KUKA KRL program: MyProgram_031().src

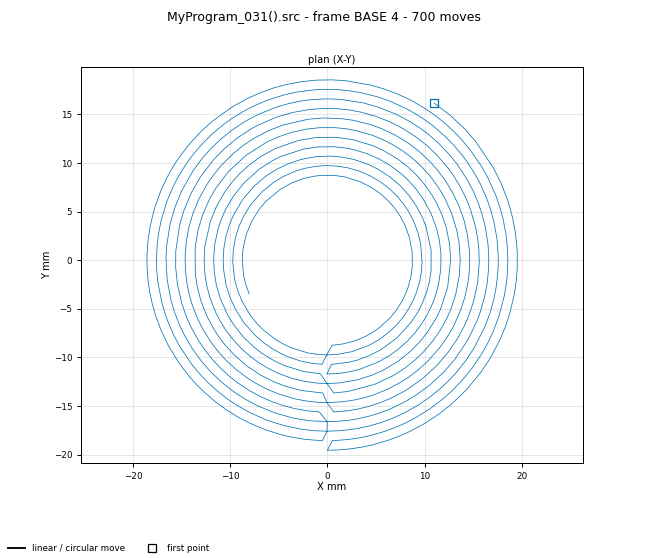
[picture p0: tool path of MyProgram_031().src in frame BASE 4, 700 of 700 moves have a stored position in this frame; points joined in program order, loops and branches not executed]
&ACCESS RVP
&REL 1
&PARAM TEMPLATE = C:\KRC\Roboter\Template\vorgabe
&PARAM EDITMASK = *
DEF MyProgram_031()
; ---- Setting reference (Base) ----
$BASE = BASE_DATA[4]

; --------------------------
; ---- Setting tool (TCP) ----
$TOOL = TOOL_DATA[3]
; --------------------------

$VEL.CP = VEL_APROX_PRINT
Startdeposition()
$VEL.CP = VEL_PRINT
LIN {X 10.9934,Y 16.1646,Z 59,A 46.5533,B 24.7923,C -3.3229,E1 25.0931,E2 -684.1777} C_DIS
LIN {X 12.5371,Y 14.9988,Z 59,A 41.0137,B 24.7934,C -3.3139,E1 25.1052,E2 -678.6373} C_DIS
LIN {X 14.028,Y 13.6149,Z 59,A 34.9278,B 24.795,C -3.3008,E1 25.1174,E2 -672.5458} C_DIS
LIN {X 15.29,Y 12.1806,Z 59,A 28.493,B 24.7975,C -3.281,E1 25.1289,E2 -666.0937} C_DIS
LIN {X 17.0834,Y 9.5029,Z 59,A 20.9449,B 24.7984,C -3.2739,E1 25.1402,E2 -658.5668} C_DIS
LIN {X 17.8595,Y 7.9485,Z 59,A 14.4237,B 24.8017,C -3.2472,E1 25.148,E2 -652.0173} C_DIS
LIN {X 18.5084,Y 6.2918,Z 59,A 10.2599,B 24.8023,C -3.2419,E1 25.152,E2 -647.8642} C_DIS
LIN {X 18.8302,Y 5.2505,Z 59,A 7.0393,B 24.8035,C -3.2323,E1 25.1545,E2 -644.6393} C_DIS
LIN {X 19.0668,Y 4.3128,Z 59,A 3.787,B 24.805,C -3.22,E1 25.1566,E2 -641.3766} C_DIS
LIN {X 19.331,Y 2.9059,Z 59,A 0.1157,B 24.806,C -3.2121,E1 25.1583,E2 -637.7083} C_DIS
LIN {X 19.4777,Y 1.6618,Z 59,A -3.1967,B 24.8069,C -3.2042,E1 25.1593,E2 -634.3968} C_DIS
LIN {X 19.5336,Y 0.7644,Z 59,A -6.4456,B 24.8086,C -3.1903,E1 25.1597,E2 -631.1341} C_DIS
LIN {X 19.5284,Y -0.889,Z 59,A -10.5652,B 24.8096,C -3.182,E1 25.1596,E2 -627.0194} C_DIS
LIN {X 19.4419,Y -2.0395,Z 59,A -14.3602,B 24.8113,C -3.1676,E1 25.1586,E2 -623.2127} C_DIS
LIN {X 19.2406,Y -3.4554,Z 59,A -19.2929,B 24.8137,C -3.1476,E1 25.1564,E2 -618.2616} C_DIS
LIN {X 18.7455,Y -5.5452,Z 59,A -24.8888,B 24.8152,C -3.1348,E1 25.1525,E2 -612.6677} C_DIS
LIN {X 18.3078,Y -6.8534,Z 59,A -28.9539,B 24.8167,C -3.1224,E1 25.1487,E2 -608.596} C_DIS
LIN {X 17.7883,Y -8.1069,Z 59,A -33.3998,B 24.8186,C -3.1064,E1 25.1437,E2 -604.1364} C_DIS
LIN {X 16.7634,Y -10.0571,Z 59,A -39.0828,B 24.8199,C -3.0952,E1 25.136,E2 -598.4565} C_DIS
LIN {X 15.7922,Y -11.5219,Z 59,A -45.0383,B 24.8223,C -3.0741,E1 25.1265,E2 -592.4803} C_DIS
LIN {X 14.2679,Y -13.3632,Z 59,A -52.0299,B 24.8243,C -3.0568,E1 25.1136,E2 -585.4791} C_DIS
LIN {X 12.7755,Y -14.7963,Z 59,A -57.4268,B 24.8253,C -3.0488,E1 25.1025,E2 -580.085} C_DIS
LIN {X 11.5072,Y -15.803,Z 59,A -62.4088,B 24.8266,C -3.037,E1 25.0914,E2 -575.0932} C_DIS
LIN {X 9.973,Y -16.8133,Z 59,A -67.5385,B 24.8275,C -3.0291,E1 25.0793,E2 -569.9612} C_DIS
LIN {X 8.5686,Y -17.5705,Z 59,A -72.3693,B 24.8285,C -3.0203,E1 25.0673,E2 -565.1228} C_DIS
LIN {X 7.4388,Y -18.0777,Z 59,A -75.5292,B 24.8287,C -3.0187,E1 25.0592,E2 -561.9667} C_DIS
LIN {X 6.3063,Y -18.5035,Z 59,A -79.4929,B 24.8296,C -3.0111,E1 25.0488,E2 -557.9929} C_DIS
LIN {X 4.7039,Y -18.9743,Z 59,A -83.9715,B 24.8298,C -3.009,E1 25.0367,E2 -553.5168} C_DIS
LIN {X 3.7008,Y -19.195,Z 59,A -86.9714,B 24.8301,C -3.0065,E1 25.0285,E2 -550.5147} C_DIS
LIN {X 2.5135,Y -19.3863,Z 59,A -90.6996,B 24.8305,C -3.0027,E1 25.0182,E2 -546.7808} C_DIS
LIN {X 1.1875,Y -19.5124,Z 59,A -94.7053,B 24.8308,C -3.0002,E1 25.007,E2 -542.7711} C_DIS
LIN {X -0.014,Y -19.5462,Z 59,A -96.7565,B 24.8298,C -3.0091,E1 25.0014,E2 -540.7413} C_DIS
Enddeposition()
LIN {X -0.014,Y -19.5462,Z 59,A -96.7565,B 24.8298,C -3.0091,E1 25.0014,E2 -540.7413} C_DIS
Startdeposition()
$VEL.CP = VEL_PRINT
LIN {X 0.5237,Y -18.5604,Z 59,A -93.787,B 24.8269,C -3.035,E1 25.0098,E2 -543.772} C_DIS
LIN {X 2.1884,Y -18.4383,Z 59,A -89.5474,B 24.8272,C -3.0316,E1 25.0216,E2 -548.0007} C_DIS
LIN {X 3.3621,Y -18.2608,Z 59,A -86.0615,B 24.8271,C -3.033,E1 25.0312,E2 -551.4866} C_DIS
LIN {X 4.4772,Y -18.0199,Z 59,A -81.9917,B 24.8263,C -3.0402,E1 25.0423,E2 -555.5678} C_DIS
LIN {X 5.9095,Y -17.6007,Z 59,A -77.975,B 24.8261,C -3.0412,E1 25.053,E2 -559.5795} C_DIS
LIN {X 7.3368,Y -17.0569,Z 59,A -73.4193,B 24.8256,C -3.0463,E1 25.0648,E2 -564.1373} C_DIS
LIN {X 8.1484,Y -16.6843,Z 59,A -70.3831,B 24.8248,C -3.0528,E1 25.0725,E2 -567.1809} C_DIS
LIN {X 9.0499,Y -16.213,Z 59,A -66.8043,B 24.8238,C -3.0616,E1 25.0813,E2 -570.7702} C_DIS
LIN {X 10.5141,Y -15.3044,Z 59,A -61.4455,B 24.8226,C -3.0719,E1 25.0938,E2 -576.1361} C_DIS
LIN {X 11.669,Y -14.4426,Z 59,A -57.2471,B 24.8218,C -3.0792,E1 25.1031,E2 -580.3362} C_DIS
LIN {X 12.719,Y -13.5275,Z 59,A -53.0786,B 24.8208,C -3.0878,E1 25.1117,E2 -584.5083} C_DIS
LIN {X 13.8411,Y -12.3769,Z 59,A -47.8137,B 24.819,C -3.1025,E1 25.1218,E2 -589.785} C_DIS
LIN {X 14.8798,Y -11.1066,Z 59,A -42.8261,B 24.8176,C -3.1149,E1 25.1303,E2 -594.7786} C_DIS
LIN {X 15.8537,Y -9.6656,Z 59,A -37.7384,B 24.8161,C -3.1271,E1 25.138,E2 -599.8697} C_DIS
LIN {X 16.5051,Y -8.5047,Z 59,A -33.7941,B 24.8149,C -3.1373,E1 25.1433,E2 -603.8175} C_DIS
LIN {X 17.0454,Y -7.3631,Z 59,A -29.7118,B 24.8134,C -3.1504,E1 25.148,E2 -607.9086} C_DIS
LIN {X 17.6434,Y -5.7852,Z 59,A -23.9683,B 24.8109,C -3.1711,E1 25.1533,E2 -613.6688} C_DIS
LIN {X 18.2032,Y -3.6604,Z 59,A -17.5312,B 24.8088,C -3.1887,E1 25.1574,E2 -620.1104} C_DIS
LIN {X 18.4301,Y -2.258,Z 59,A -13.7246,B 24.8078,C -3.197,E1 25.1589,E2 -623.9142} C_DIS
LIN {X 18.5284,Y -1.2107,Z 59,A -10.5836,B 24.8067,C -3.2061,E1 25.1596,E2 -627.0582} C_DIS
LIN {X 18.5698,Y -0.0273,Z 59,A -6.3825,B 24.8047,C -3.2226,E1 25.1597,E2 -631.2734} C_DIS
LIN {X 18.5205,Y 1.3276,Z 59,A -2.3554,B 24.8033,C -3.2341,E1 25.1591,E2 -635.3039} C_DIS
LIN {X 18.3716,Y 2.6925,Z 59,A 1.9622,B 24.8016,C -3.2478,E1 25.1575,E2 -639.6284} C_DIS
LIN {X 18.075,Y 4.2502,Z 59,A 6.671,B 24.8,C -3.2608,E1 25.1548,E2 -644.3406} C_DIS
LIN {X 17.7604,Y 5.4158,Z 59,A 10.2503,B 24.7988,C -3.2704,E1 25.152,E2 -647.9222} C_DIS
LIN {X 17.3583,Y 6.5919,Z 59,A 14.5526,B 24.7969,C -3.2855,E1 25.1478,E2 -652.2364} C_DIS
LIN {X 16.5083,Y 8.4991,Z 59,A 20.2918,B 24.7955,C -3.2968,E1 25.141,E2 -657.9714} C_DIS
LIN {X 15.8062,Y 9.7434,Z 59,A 25.4816,B 24.7933,C -3.315,E1 25.1335,E2 -663.1777} C_DIS
LIN {X 14.5876,Y 11.4876,Z 59,A 31.3946,B 24.792,C -3.325,E1 25.1238,E2 -669.0861} C_DIS
LIN {X 13.6613,Y 12.575,Z 59,A 35.618,B 24.791,C -3.3332,E1 25.116,E2 -673.3099} C_DIS
LIN {X 12.7974,Y 13.4532,Z 59,A 39.7636,B 24.7896,C -3.3437,E1 25.1077,E2 -677.4632} C_DIS
LIN {X 11.9589,Y 14.2042,Z 59,A 43.058,B 24.789,C -3.3488,E1 25.1007,E2 -680.7568} C_DIS
LIN {X 11.0207,Y 14.9437,Z 59,A 46.3495,B 24.7886,C -3.3521,E1 25.0934,E2 -684.0441} C_DIS
LIN {X 9.9784,Y 15.6588,Z 59,A 50.7011,B 24.7874,C -3.3616,E1 25.0833,E2 -688.4039} C_DIS
LIN {X 8.6913,Y 16.4082,Z 59,A 55.2475,B 24.7866,C -3.3674,E1 25.0722,E2 -692.9507} C_DIS
LIN {X 7.4621,Y 17.0024,Z 59,A 59.3101,B 24.7862,C -3.371,E1 25.0619,E2 -697.0117} C_DIS
LIN {X 5.9289,Y 17.5955,Z 59,A 64.5931,B 24.7854,C -3.377,E1 25.048,E2 -702.2978} C_DIS
LIN {X 4.4746,Y 18.0207,Z 59,A 69.9369,B 24.7845,C -3.3843,E1 25.0335,E2 -707.6509} C_DIS
LIN {X 1.7966,Y 18.4808,Z 59,A 77.036,B 24.7852,C -3.3783,E1 25.014,E2 -714.7291} C_DIS
LIN {X 0.4664,Y 18.562,Z 59,A 81.8933,B 24.7847,C -3.3825,E1 25.0004,E2 -719.5951} C_DIS
LIN {X -1.1715,Y 18.5307,Z 59,A 86.5563,B 24.7852,C -3.3787,E1 24.9874,E2 -724.2497} C_DIS
LIN {X -2.6397,Y 18.3778,Z 59,A 90.8462,B 24.7857,C -3.3747,E1 24.9756,E2 -728.533} C_DIS
LIN {X -4.1478,Y 18.0986,Z 59,A 96.1737,B 24.7857,C -3.374,E1 24.961,E2 -733.865} C_DIS
LIN {X -5.4949,Y 17.7361,Z 59,A 100.4335,B 24.7864,C -3.3692,E1 24.9496,E2 -738.1204} C_DIS
LIN {X -7.0138,Y 17.1921,Z 59,A 105.1464,B 24.7874,C -3.3615,E1 24.9373,E2 -742.8249} C_DIS
LIN {X -8.3436,Y 16.5877,Z 59,A 110.1725,B 24.7879,C -3.3571,E1 24.9246,E2 -747.8532} C_DIS
LIN {X -9.8622,Y 15.7322,Z 59,A 115.7778,B 24.789,C -3.3486,E1 24.9112,E2 -753.4554} C_DIS
LIN {X -11.794,Y 14.3412,Z 59,A 122.0514,B 24.7915,C -3.3294,E1 24.8973,E2 -759.7053} C_DIS
LIN {X -12.9768,Y 13.2796,Z 59,A 128.0289,B 24.7923,C -3.3224,E1 24.885,E2 -765.6906} C_DIS
LIN {X -14.3419,Y 11.7922,Z 59,A 134.5147,B 24.7941,C -3.3079,E1 24.8732,E2 -772.1711} C_DIS
LIN {X -15.524,Y 10.1868,Z 59,A 139.7208,B 24.7966,C -3.2883,E1 24.8649,E2 -777.3557} C_DIS
LIN {X -16.0114,Y 9.4022,Z 59,A 142.6599,B 24.7975,C -3.2807,E1 24.8607,E2 -780.2918} C_DIS
LIN {X -16.5699,Y 8.3788,Z 59,A 146.5868,B 24.7987,C -3.2715,E1 24.8556,E2 -784.2176} C_DIS
LIN {X -17.1414,Y 7.1369,Z 59,A 150.9696,B 24.8001,C -3.2597,E1 24.8507,E2 -788.5962} C_DIS
LIN {X -17.7821,Y 5.3442,Z 59,A 157.1224,B 24.8022,C -3.2429,E1 24.8454,E2 -794.7439} C_DIS
LIN {X -18.2292,Y 3.5294,Z 59,A 162.1023,B 24.8047,C -3.2227,E1 24.8423,E2 -799.7047} C_DIS
LIN {X -18.4463,Y 2.1199,Z 59,A 167.1635,B 24.8061,C -3.211,E1 24.8404,E2 -804.7681} C_DIS
LIN {X -18.5634,Y 0.4029,Z 59,A 172.0002,B 24.8083,C -3.1931,E1 24.8398,E2 -809.5908} C_DIS
LIN {X -18.5529,Y -0.7461,Z 59,A 175.4062,B 24.8096,C -3.1816,E1 24.84,E2 -812.99} C_DIS
LIN {X -18.4568,Y -2.027,Z 59,A 179.3572,B 24.8111,C -3.1694,E1 24.8409,E2 -816.9354} C_DIS
LIN {X -18.3051,Y -3.1127,Z 59,A -176.6587,B 24.8121,C -3.161,E1 24.8427,E2 -820.923} C_DIS
LIN {X -18.0102,Y -4.5166,Z 59,A -172.3898,B 24.8137,C -3.1473,E1 24.8453,E2 -825.1841} C_DIS
LIN {X -17.6745,Y -5.69,Z 59,A -168.215,B 24.8149,C -3.1377,E1 24.8488,E2 -829.3599} C_DIS
LIN {X -17.09,Y -7.2591,Z 59,A -163.1852,B 24.8167,C -3.1227,E1 24.854,E2 -834.3819} C_DIS
LIN {X -16.3676,Y -8.7671,Z 59,A -158.089,B 24.8183,C -3.1086,E1 24.8604,E2 -839.4719} C_DIS
LIN {X -15.3002,Y -10.52,Z 59,A -150.8716,B 24.8198,C -3.0961,E1 24.8713,E2 -846.6957} C_DIS
LIN {X -14.1699,Y -11.9992,Z 59,A -146.4366,B 24.8219,C -3.0779,E1 24.879,E2 -851.1077} C_DIS
LIN {X -13.5514,Y -12.6934,Z 59,A -142.9303,B 24.8223,C -3.0743,E1 24.8857,E2 -854.6209} C_DIS
LIN {X -12.6198,Y -13.6202,Z 59,A -138.756,B 24.8232,C -3.0667,E1 24.8941,E2 -858.7944} C_DIS
LIN {X -11.4375,Y -14.6271,Z 59,A -134.7068,B 24.8246,C -3.0549,E1 24.9028,E2 -862.8306} C_DIS
LIN {X -10.4429,Y -15.3528,Z 59,A -130.1092,B 24.8249,C -3.0524,E1 24.9133,E2 -867.438} C_DIS
LIN {X -9.2262,Y -16.1134,Z 59,A -126.1346,B 24.8258,C -3.044,E1 24.9228,E2 -871.4047} C_DIS
LIN {X -8.0735,Y -16.7207,Z 59,A -121.9508,B 24.8263,C -3.04,E1 24.9333,E2 -875.5902} C_DIS
LIN {X -6.4151,Y -17.4242,Z 59,A -115.4888,B 24.8263,C -3.0396,E1 24.9501,E2 -882.0652} C_DIS
LIN {X -4.7827,Y -17.9413,Z 59,A -111.2767,B 24.8274,C -3.0302,E1 24.9613,E2 -886.2617} C_DIS
LIN {X -3.7911,Y -18.1762,Z 59,A -108.016,B 24.8274,C -3.0294,E1 24.9702,E2 -889.5247} C_DIS
LIN {X -2.2382,Y -18.4325,Z 59,A -102.9506,B 24.8274,C -3.0296,E1 24.9842,E2 -894.5947} C_DIS
LIN {X -0.5182,Y -18.5594,Z 59,A -97.8029,B 24.8276,C -3.0288,E1 24.9986,E2 -899.742} C_DIS
LIN {X -0.5182,Y -18.5594,Z 59,A -97.8029,B 24.8276,C -3.0288,E1 24.9986,E2 -899.742} C_DIS
Enddeposition()
LIN {X -0.0341,Y -17.5871,Z 59,A -98.1601,B 24.8269,C -3.0347,E1 24.9976,E2 -899.3987} C_DIS
Startdeposition()
$VEL.CP = VEL_PRINT
LIN {X -1.202,Y -17.546,Z 59,A -102.1315,B 24.827,C -3.0335,E1 24.9865,E2 -895.4234} C_DIS
LIN {X -2.6082,Y -17.3925,Z 59,A -107.1397,B 24.8272,C -3.0321,E1 24.9726,E2 -890.4083} C_DIS
LIN {X -4.5044,Y -17.0004,Z 59,A -113.0275,B 24.8266,C -3.0373,E1 24.9566,E2 -884.5252} C_DIS
LIN {X -6.2144,Y -16.4525,Z 59,A -119.7875,B 24.8266,C -3.0376,E1 24.9388,E2 -877.753} C_DIS
LIN {X -7.9886,Y -15.6679,Z 59,A -125.5503,B 24.8254,C -3.0473,E1 24.9243,E2 -871.9985} C_DIS
LIN {X -9.3669,Y -14.8852,Z 59,A -130.316,B 24.8244,C -3.0562,E1 24.9129,E2 -867.2397} C_DIS
LIN {X -10.2976,Y -14.2571,Z 59,A -133.7611,B 24.8236,C -3.0629,E1 24.905,E2 -863.7988} C_DIS
LIN {X -11.2418,Y -13.5251,Z 59,A -138.3974,B 24.8232,C -3.0669,E1 24.8949,E2 -859.1548} C_DIS
LIN {X -12.4133,Y -12.4588,Z 59,A -143.1705,B 24.8218,C -3.0785,E1 24.8852,E2 -854.3898} C_DIS
LIN {X -13.276,Y -11.5347,Z 59,A -147.4681,B 24.8209,C -3.0868,E1 24.8772,E2 -850.093} C_DIS
LIN {X -14.0207,Y -10.6174,Z 59,A -152.0625,B 24.8201,C -3.0934,E1 24.8693,E2 -845.4924} C_DIS
LIN {X -15.21,Y -8.8298,Z 59,A -158.0938,B 24.8177,C -3.1139,E1 24.8604,E2 -839.4797} C_DIS
LIN {X -15.8554,Y -7.6095,Z 59,A -162.9618,B 24.8164,C -3.1249,E1 24.8542,E2 -834.6118} C_DIS
LIN {X -16.5043,Y -6.0742,Z 59,A -169.1979,B 24.8149,C -3.1379,E1 24.8479,E2 -828.3721} C_DIS
LIN {X -16.9974,Y -4.5159,Z 59,A -174.5907,B 24.813,C -3.1534,E1 24.8438,E2 -822.985} C_DIS
LIN {X -17.4451,Y -2.2294,Z 59,A 179.1035,B 24.8099,C -3.1797,E1 24.8409,E2 -816.7048} C_DIS
LIN {X -17.5572,Y -1.0226,Z 59,A 175.2609,B 24.8084,C -3.1921,E1 24.84,E2 -812.8688} C_DIS
LIN {X -17.5889,Y -0.0438,Z 59,A 170.9905,B 24.8075,C -3.1993,E1 24.8398,E2 -808.59} C_DIS
LIN {X -17.5028,Y 1.7202,Z 59,A 165.8261,B 24.8052,C -3.2187,E1 24.8408,E2 -803.441} C_DIS
LIN {X -17.3482,Y 2.8889,Z 59,A 161.8878,B 24.8037,C -3.2303,E1 24.8424,E2 -799.5072} C_DIS
LIN {X -17.1003,Y 4.1084,Z 59,A 157.2587,B 24.8024,C -3.2414,E1 24.8453,E2 -794.8774} C_DIS
LIN {X -16.5111,Y 6.057,Z 59,A 150.2732,B 24.8,C -3.2604,E1 24.8515,E2 -787.8977} C_DIS
LIN {X -15.838,Y 7.646,Z 59,A 145.3885,B 24.7978,C -3.2787,E1 24.8571,E2 -783.0302} C_DIS
LIN {X -15.2784,Y 8.7108,Z 59,A 141.3244,B 24.7965,C -3.2894,E1 24.8625,E2 -778.9702} C_DIS
LIN {X -14.5545,Y 9.8727,Z 59,A 137.2092,B 24.7948,C -3.3025,E1 24.8688,E2 -774.8656} C_DIS
LIN {X -13.9706,Y 10.683,Z 59,A 133.478,B 24.7939,C -3.3095,E1 24.875,E2 -771.1334} C_DIS
LIN {X -13,Y 11.8452,Z 59,A 128.5098,B 24.7924,C -3.3216,E1 24.8841,E2 -766.1716} C_DIS
LIN {X -11.8535,Y 12.9918,Z 59,A 123.7688,B 24.7907,C -3.3355,E1 24.8936,E2 -761.4442} C_DIS
LIN {X -10.7852,Y 13.892,Z 59,A 119.0842,B 24.7895,C -3.3447,E1 24.9037,E2 -756.7638} C_DIS
LIN {X -9.7714,Y 14.623,Z 59,A 114.5567,B 24.7887,C -3.3509,E1 24.9141,E2 -752.2359} C_DIS
LIN {X -8.6558,Y 15.3098,Z 59,A 110.5552,B 24.7877,C -3.3594,E1 24.9237,E2 -748.2425} C_DIS
LIN {X -7.5105,Y 15.9027,Z 59,A 106.0225,B 24.787,C -3.3646,E1 24.935,E2 -743.7103} C_DIS
LIN {X -6.2319,Y 16.4459,Z 59,A 101.4023,B 24.7863,C -3.3702,E1 24.947,E2 -739.0934} C_DIS
LIN {X -4.4803,Y 17.0067,Z 59,A 96.1433,B 24.785,C -3.3799,E1 24.961,E2 -733.8488} C_DIS
LIN {X -3.1544,Y 17.3018,Z 59,A 90.8771,B 24.785,C -3.3795,E1 24.9754,E2 -728.5754} C_DIS
LIN {X -1.3631,Y 17.534,Z 59,A 85.5279,B 24.7843,C -3.3853,E1 24.9903,E2 -723.2369} C_DIS
LIN {X -0.2748,Y 17.585,Z 59,A 81.8951,B 24.7843,C -3.3859,E1 25.0004,E2 -719.605} C_DIS
LIN {X 0.9445,Y 17.5616,Z 59,A 77.9768,B 24.7842,C -3.3865,E1 25.0113,E2 -715.6891} C_DIS
LIN {X 2.0251,Y 17.4701,Z 59,A 74.5767,B 24.7842,C -3.3869,E1 25.0208,E2 -712.292} C_DIS
LIN {X 3.3851,Y 17.2583,Z 59,A 69.3654,B 24.7849,C -3.381,E1 25.0351,E2 -707.0723} C_DIS
LIN {X 5.1414,Y 16.8186,Z 59,A 63.7363,B 24.7852,C -3.3789,E1 25.0503,E2 -701.4474} C_DIS
LIN {X 6.5268,Y 16.3312,Z 59,A 58.7341,B 24.7859,C -3.3731,E1 25.0633,E2 -696.4421} C_DIS
LIN {X 8.2661,Y 15.5236,Z 59,A 52.7014,B 24.7867,C -3.3671,E1 25.0784,E2 -690.4112} C_DIS
LIN {X 9.239,Y 14.9649,Z 59,A 49.4605,B 24.787,C -3.3648,E1 25.0862,E2 -687.1748} C_DIS
LIN {X 10.1074,Y 14.3927,Z 59,A 46.1864,B 24.7875,C -3.3602,E1 25.0937,E2 -683.901} C_DIS
LIN {X 10.8842,Y 13.8142,Z 59,A 42.5638,B 24.7887,C -3.3513,E1 25.1018,E2 -680.2704} C_DIS
LIN {X 12.1818,Y 12.685,Z 59,A 36.9397,B 24.7901,C -3.3402,E1 25.1134,E2 -674.6427} C_DIS
LIN {X 13.0558,Y 11.7832,Z 59,A 33.0738,B 24.791,C -3.3332,E1 25.1207,E2 -670.7771} C_DIS
LIN {X 13.8849,Y 10.7944,Z 59,A 29.1416,B 24.7919,C -3.3258,E1 25.1276,E2 -666.8454} C_DIS
LIN {X 14.4707,Y 9.9948,Z 59,A 25.5134,B 24.7933,C -3.3147,E1 25.1335,E2 -663.2087} C_DIS
LIN {X 15.296,Y 8.6798,Z 59,A 20.8881,B 24.7945,C -3.3053,E1 25.1402,E2 -658.5848} C_DIS
LIN {X 15.7748,Y 7.7754,Z 59,A 17.229,B 24.7959,C -3.2937,E1 25.1448,E2 -654.9175} C_DIS
LIN {X 16.3754,Y 6.4149,Z 59,A 12.8077,B 24.7972,C -3.2837,E1 25.1496,E2 -650.4969} C_DIS
LIN {X 16.7585,Y 5.3277,Z 59,A 9.1385,B 24.7984,C -3.2737,E1 25.1529,E2 -646.8246} C_DIS
LIN {X 17.1612,Y 3.847,Z 59,A 3.5488,B 24.8009,C -3.2537,E1 25.1567,E2 -641.2198} C_DIS
LIN {X 17.4561,Y 2.1435,Z 59,A -2.1885,B 24.8031,C -3.2357,E1 25.159,E2 -635.4734} C_DIS
LIN {X 17.5829,Y 0.389,Z 59,A -7.321,B 24.8046,C -3.2232,E1 25.1598,E2 -630.3418} C_DIS
LIN {X 17.5693,Y -0.791,Z 59,A -11.7704,B 24.8067,C -3.2059,E1 25.1594,E2 -625.8779} C_DIS
LIN {X 17.3971,Y -2.5796,Z 59,A -17.0839,B 24.8083,C -3.1924,E1 25.1576,E2 -620.5638} C_DIS
LIN {X 17.1448,Y -3.9184,Z 59,A -21.4856,B 24.81,C -3.179,E1 25.1551,E2 -616.156} C_DIS
LIN {X 16.7502,Y -5.3608,Z 59,A -26.9183,B 24.8123,C -3.1593,E1 25.1507,E2 -610.7076} C_DIS
LIN {X 16.2207,Y -6.7963,Z 59,A -32.3118,B 24.8145,C -3.141,E1 25.1451,E2 -605.3005} C_DIS
LIN {X 15.1393,Y -8.9502,Z 59,A -39.1864,B 24.8162,C -3.127,E1 25.136,E2 -598.4287} C_DIS
LIN {X 14.2994,Y -10.2387,Z 59,A -43.7759,B 24.8173,C -3.1169,E1 25.1288,E2 -593.8382} C_DIS
LIN {X 13.3413,Y -11.4595,Z 59,A -48.9758,B 24.819,C -3.1028,E1 25.1196,E2 -588.6289} C_DIS
LIN {X 12.4978,Y -12.3738,Z 59,A -53.1294,B 24.8202,C -3.0922,E1 25.1116,E2 -584.4683} C_DIS
LIN {X 11.523,Y -13.2864,Z 59,A -57.5824,B 24.8215,C -3.0816,E1 25.1024,E2 -580.0079} C_DIS
LIN {X 10.5304,Y -14.0857,Z 59,A -61.3966,B 24.8222,C -3.0756,E1 25.0939,E2 -576.1935} C_DIS
LIN {X 9.3514,Y -14.8949,Z 59,A -66.5114,B 24.8236,C -3.0633,E1 25.082,E2 -571.0663} C_DIS
LIN {X 7.881,Y -15.7225,Z 59,A -71.8747,B 24.8245,C -3.0551,E1 25.0688,E2 -565.6989} C_DIS
LIN {X 6.6785,Y -16.2696,Z 59,A -75.7384,B 24.8249,C -3.052,E1 25.0589,E2 -561.8372} C_DIS
LIN {X 5.5387,Y -16.6921,Z 59,A -79.5762,B 24.8254,C -3.0479,E1 25.0488,E2 -557.9973} C_DIS
LIN {X 4.3173,Y -17.049,Z 59,A -84.2933,B 24.8263,C -3.0397,E1 25.036,E2 -553.2684} C_DIS
LIN {X 3.067,Y -17.3175,Z 59,A -88.4641,B 24.8267,C -3.0363,E1 25.0246,E2 -549.0944} C_DIS
LIN {X 1.512,Y -17.5221,Z 59,A -93.4732,B 24.827,C -3.0341,E1 25.0107,E2 -544.0834} C_DIS
LIN {X -0.0341,Y -17.5871,Z 59,A -95.9822,B 24.8254,C -3.0478,E1 25.0038,E2 -541.6078} C_DIS
Enddeposition()
LIN {X -0.0167,Y -16.6038,Z 59,A -2.603,B -0.0001,C -0.0021,E1 0.1598,E2 -630.6872} C_DIS
Startdeposition()
$VEL.CP = VEL_PRINT
LIN {X 0.9904,Y -16.5764,Z 59,A -2.567,B -0.0002,C -0.0021,E1 0.1597,E2 -630.6857} C_DIS
LIN {X 2.1202,Y -16.4703,Z 59,A -2.5264,B -0.0004,C -0.0021,E1 0.1595,E2 -630.681} C_DIS
LIN {X 3.0555,Y -16.3228,Z 59,A -2.4952,B -0.0005,C -0.0021,E1 0.1594,E2 -630.6719} C_DIS
LIN {X 4.3685,Y -16.0213,Z 59,A -2.4467,B -0.0007,C -0.0021,E1 0.1592,E2 -630.6599} C_DIS
LIN {X 5.3661,Y -15.7154,Z 59,A -2.4124,B -0.0007,C -0.002,E1 0.1591,E2 -630.6448} C_DIS
LIN {X 6.4776,Y -15.2909,Z 59,A -2.3767,B -0.001,C -0.0019,E1 0.1589,E2 -630.6217} C_DIS
LIN {X 7.9833,Y -14.5611,Z 59,A -2.3219,B -0.0011,C -0.0018,E1 0.1587,E2 -630.59} C_DIS
LIN {X 9.1663,Y -13.8473,Z 59,A -2.2799,B -0.0013,C -0.0017,E1 0.1587,E2 -630.5578} C_DIS
LIN {X 10.5664,Y -12.8103,Z 59,A -2.2377,B -0.0015,C -0.0015,E1 0.1584,E2 -630.5035} C_DIS
LIN {X 12.0029,Y -11.4754,Z 59,A -2.1921,B -0.0016,C -0.0013,E1 0.1582,E2 -630.438} C_DIS
LIN {X 13.1246,Y -10.1742,Z 59,A -2.1569,B -0.0018,C -0.0012,E1 0.1581,E2 -630.375} C_DIS
LIN {X 14.4222,Y -8.2322,Z 59,A -2.1137,B -0.0019,C -0.0009,E1 0.1579,E2 -630.2853} C_DIS
LIN {X 15.3466,Y -6.3442,Z 59,A -2.0661,B -0.0019,C -0.0007,E1 0.1579,E2 -630.2164} C_DIS
LIN {X 15.729,Y -5.3263,Z 59,A -2.0674,B -0.002,C -0.0006,E1 0.1578,E2 -630.1562} C_DIS
LIN {X 16.1828,Y -3.7261,Z 59,A -2.0525,B -0.002,C -0.0004,E1 0.1578,E2 -630.0842} C_DIS
LIN {X 16.4301,Y -2.4133,Z 59,A -2.0455,B -0.0021,C -0.0002,E1 0.1577,E2 -630.0246} C_DIS
LIN {X 16.5743,Y -1.0125,Z 59,A -2.0396,B -0.0021,C 0,E1 0.1577,E2 -629.964} C_DIS
LIN {X 16.6055,Y 0.1927,Z 59,A -2.046,B -0.0021,C 0.0001,E1 0.1577,E2 -629.9038} C_DIS
LIN {X 16.5283,Y 1.6086,Z 59,A -2.0584,B -0.0021,C 0.0003,E1 0.1577,E2 -629.8325} C_DIS
LIN {X 16.2604,Y 3.3713,Z 59,A -2.0679,B -0.0021,C 0.0005,E1 0.1577,E2 -629.7563} C_DIS
LIN {X 15.9251,Y 4.7056,Z 59,A -2.0806,B -0.002,C 0.0007,E1 0.1577,E2 -629.6984} C_DIS
LIN {X 15.4863,Y 5.9956,Z 59,A -2.106,B -0.002,C 0.0009,E1 0.1578,E2 -629.6335} C_DIS
LIN {X 15.0367,Y 7.0473,Z 59,A -2.1262,B -0.0019,C 0.001,E1 0.1579,E2 -629.5847} C_DIS
LIN {X 14.3539,Y 8.3512,Z 59,A -2.1566,B -0.0018,C 0.0012,E1 0.1579,E2 -629.5237} C_DIS
LIN {X 13.351,Y 9.8748,Z 59,A -2.1863,B -0.0016,C 0.0013,E1 0.1581,E2 -629.4663} C_DIS
LIN {X 12.5968,Y 10.821,Z 59,A -2.227,B -0.0016,C 0.0015,E1 0.1582,E2 -629.4133} C_DIS
LIN {X 11.4808,Y 11.9985,Z 59,A -2.2698,B -0.0014,C 0.0016,E1 0.1584,E2 -629.3622} C_DIS
LIN {X 10.3808,Y 12.962,Z 59,A -2.3081,B -0.0012,C 0.0017,E1 0.1584,E2 -629.3243} C_DIS
LIN {X 9.587,Y 13.5597,Z 59,A -2.3443,B -0.0012,C 0.0018,E1 0.1586,E2 -629.2926} C_DIS
LIN {X 8.5013,Y 14.2653,Z 59,A -2.3855,B -0.001,C 0.0018,E1 0.1588,E2 -629.2625} C_DIS
LIN {X 7.0867,Y 15.0181,Z 59,A -2.4413,B -0.0008,C 0.002,E1 0.159,E2 -629.2281} C_DIS
LIN {X 5.2232,Y 15.7634,Z 59,A -2.5104,B -0.0005,C 0.002,E1 0.1592,E2 -629.198} C_DIS
LIN {X 3.6139,Y 16.2079,Z 59,A -2.5708,B -0.0003,C 0.002,E1 0.1594,E2 -629.1796} C_DIS
LIN {X 1.3286,Y 16.5531,Z 59,A -2.6524,B 0,C 0.0021,E1 0.1597,E2 -629.1697} C_DIS
LIN {X -0.0236,Y 16.6065,Z 59,A -2.7012,B 0.0002,C 0.0021,E1 0.1599,E2 -629.1697} C_DIS
LIN {X -1.5553,Y 16.5333,Z 59,A -2.7565,B 0.0003,C 0.0021,E1 0.16,E2 -629.1751} C_DIS
LIN {X -2.7667,Y 16.3742,Z 59,A -2.7997,B 0.0005,C 0.0021,E1 0.1602,E2 -629.1841} C_DIS
LIN {X -3.9498,Y 16.1297,Z 59,A -2.8411,B 0.0006,C 0.0021,E1 0.1603,E2 -629.1973} C_DIS
LIN {X -5.2286,Y 15.7615,Z 59,A -2.8832,B 0.0008,C 0.002,E1 0.1605,E2 -629.2184} C_DIS
LIN {X -7.1262,Y 14.9994,Z 59,A -2.9471,B 0.0011,C 0.0018,E1 0.1608,E2 -629.2574} C_DIS
LIN {X -8.4091,Y 14.3198,Z 59,A -2.993,B 0.0012,C 0.0018,E1 0.1609,E2 -629.2876} C_DIS
LIN {X -9.7953,Y 13.4097,Z 59,A -3.0364,B 0.0014,C 0.0016,E1 0.1611,E2 -629.3336} C_DIS
LIN {X -11.0607,Y 12.3867,Z 59,A -3.0781,B 0.0015,C 0.0015,E1 0.1613,E2 -629.3814} C_DIS
LIN {X -12.126,Y 11.3435,Z 59,A -3.1185,B 0.0016,C 0.0013,E1 0.1613,E2 -629.424} C_DIS
LIN {X -12.8622,Y 10.5035,Z 59,A -3.1341,B 0.0017,C 0.0013,E1 0.1615,E2 -629.4704} C_DIS
LIN {X -13.8438,Y 9.1716,Z 59,A -3.1593,B 0.0019,C 0.001,E1 0.1616,E2 -629.5367} C_DIS
LIN {X -15.0107,Y 7.1025,Z 59,A -3.1988,B 0.0019,C 0.0008,E1 0.1617,E2 -629.6261} C_DIS
LIN {X -15.7152,Y 5.3667,Z 59,A -3.2115,B 0.0021,C 0.0005,E1 0.1618,E2 -629.7112} C_DIS
LIN {X -16.1915,Y 3.6878,Z 59,A -3.2212,B 0.0021,C 0.0003,E1 0.1618,E2 -629.7887} C_DIS
LIN {X -16.5438,Y 1.437,Z 59,A -3.2403,B 0.0021,C 0,E1 0.1619,E2 -629.8763} C_DIS
LIN {X -16.6045,Y 0.2489,Z 59,A -3.2246,B 0.0021,C -0.0002,E1 0.1619,E2 -629.9436} C_DIS
LIN {X -16.4836,Y -2.0164,Z 59,A -3.2086,B 0.0021,C -0.0005,E1 0.1619,E2 -630.0497} C_DIS
LIN {X -16.0863,Y -4.1232,Z 59,A -3.2036,B 0.0021,C -0.0007,E1 0.1619,E2 -630.1286} C_DIS
LIN {X -15.7744,Y -5.1895,Z 59,A -3.1849,B 0.002,C -0.0008,E1 0.1618,E2 -630.1807} C_DIS
LIN {X -15.2365,Y -6.6046,Z 59,A -3.1653,B 0.0019,C -0.001,E1 0.1618,E2 -630.2404} C_DIS
LIN {X -14.7296,Y -7.6681,Z 59,A -3.1461,B 0.0019,C -0.0011,E1 0.1617,E2 -630.2861} C_DIS
LIN {X -13.908,Y -9.074,Z 59,A -3.1038,B 0.0017,C -0.0013,E1 0.1615,E2 -630.3581} C_DIS
LIN {X -12.9961,Y -10.3379,Z 59,A -3.0716,B 0.0016,C -0.0014,E1 0.1615,E2 -630.4109} C_DIS
LIN {X -12.0357,Y -11.4418,Z 59,A -3.0367,B 0.0014,C -0.0016,E1 0.1613,E2 -630.458} C_DIS
LIN {X -10.8435,Y -12.5767,Z 59,A -2.9901,B 0.0013,C -0.0017,E1 0.1611,E2 -630.5101} C_DIS
LIN {X -9.6701,Y -13.5004,Z 59,A -2.9454,B 0.0011,C -0.0018,E1 0.161,E2 -630.5519} C_DIS
LIN {X -8.4838,Y -14.2755,Z 59,A -2.9022,B 0.0009,C -0.0018,E1 0.1608,E2 -630.5856} C_DIS
LIN {X -7.2507,Y -14.9399,Z 59,A -2.8567,B 0.0008,C -0.002,E1 0.1607,E2 -630.6153} C_DIS
LIN {X -5.4913,Y -15.6721,Z 59,A -2.7899,B 0.0005,C -0.002,E1 0.1604,E2 -630.6503} C_DIS
LIN {X -3.7975,Y -16.1648,Z 59,A -2.7331,B 0.0004,C -0.002,E1 0.1603,E2 -630.6674} C_DIS
LIN {X -2.7555,Y -16.3761,Z 59,A -2.6949,B 0.0002,C -0.0021,E1 0.1601,E2 -630.6774} C_DIS
LIN {X -1.6353,Y -16.5256,Z 59,A -2.6548,B 0.0001,C -0.0021,E1 0.16,E2 -630.6836} C_DIS
LIN {X -0.0167,Y -16.6038,Z 59,A -2.5969,B -0.0001,C -0.0021,E1 0.1598,E2 -630.6867} C_DIS
Enddeposition()
LIN {X -0.0167,Y -16.6038,Z 59,A -2.5969,B -0.0001,C -0.0021,E1 0.1598,E2 -630.6867} C_DIS
Startdeposition()
$VEL.CP = VEL_PRINT
LIN {X -0.8365,Y -15.6031,Z 59,A -2.5752,B 0.0001,C -0.0021,E1 0.16,E2 -630.6942} C_DIS
LIN {X -2.0793,Y -15.4866,Z 59,A -2.6239,B 0.0002,C -0.0021,E1 0.1601,E2 -630.6852} C_DIS
LIN {X -3.4213,Y -15.2464,Z 59,A -2.673,B 0.0004,C -0.0021,E1 0.1603,E2 -630.6739} C_DIS
LIN {X -4.4197,Y -14.9875,Z 59,A -2.7127,B 0.0005,C -0.0021,E1 0.1604,E2 -630.659} C_DIS
LIN {X -5.5531,Y -14.6054,Z 59,A -2.758,B 0.0007,C -0.0021,E1 0.1606,E2 -630.638} C_DIS
LIN {X -6.8076,Y -14.0647,Z 59,A -2.8065,B 0.0009,C -0.002,E1 0.1608,E2 -630.6113} C_DIS
LIN {X -7.9948,Y -13.4253,Z 59,A -2.8587,B 0.0011,C -0.0019,E1 0.1609,E2 -630.5743} C_DIS
LIN {X -9.1231,Y -12.6858,Z 59,A -2.902,B 0.0011,C -0.0018,E1 0.1611,E2 -630.5401} C_DIS
LIN {X -10.0197,Y -11.9902,Z 59,A -2.9405,B 0.0013,C -0.0017,E1 0.1612,E2 -630.5041} C_DIS
LIN {X -10.8903,Y -11.2055,Z 59,A -2.98,B 0.0015,C -0.0016,E1 0.1613,E2 -630.4625} C_DIS
LIN {X -11.8306,Y -10.2076,Z 59,A -3.0202,B 0.0015,C -0.0014,E1 0.1614,E2 -630.4138} C_DIS
LIN {X -12.707,Y -9.0935,Z 59,A -3.0619,B 0.0017,C -0.0013,E1 0.1616,E2 -630.3565} C_DIS
LIN {X -13.3249,Y -8.1614,Z 59,A -3.0891,B 0.0017,C -0.0012,E1 0.1616,E2 -630.3122} C_DIS
LIN {X -13.997,Y -6.9453,Z 59,A -3.1227,B 0.0019,C -0.001,E1 0.1617,E2 -630.2515} C_DIS
LIN {X -14.5067,Y -5.8063,Z 59,A -3.1431,B 0.0019,C -0.0009,E1 0.1617,E2 -630.2017} C_DIS
LIN {X -14.9859,Y -4.4244,Z 59,A -3.1875,B 0.002,C -0.0006,E1 0.1619,E2 -630.1167} C_DIS
LIN {X -15.4335,Y -2.4391,Z 59,A -3.2009,B 0.0021,C -0.0004,E1 0.1619,E2 -630.0361} C_DIS
LIN {X -15.6083,Y -0.7284,Z 59,A -3.2373,B 0.0021,C -0.0001,E1 0.1619,E2 -629.9348} C_DIS
LIN {X -15.5966,Y 0.9527,Z 59,A -3.2485,B 0.0021,C 0.0001,E1 0.1619,E2 -629.853} C_DIS
LIN {X -15.208,Y 3.5884,Z 59,A -3.2273,B 0.0021,C 0.0004,E1 0.1619,E2 -629.7499} C_DIS
LIN {X -14.7739,Y 5.0879,Z 59,A -3.2422,B 0.0021,C 0.0007,E1 0.1618,E2 -629.657} C_DIS
LIN {X -14.0035,Y 6.9318,Z 59,A -3.2187,B 0.0019,C 0.0009,E1 0.1617,E2 -629.5755} C_DIS
LIN {X -13.047,Y 8.5984,Z 59,A -3.2009,B 0.0019,C 0.0011,E1 0.1615,E2 -629.489} C_DIS
LIN {X -11.6729,Y 10.3876,Z 59,A -3.145,B 0.0017,C 0.0014,E1 0.1614,E2 -629.4194} C_DIS
LIN {X -10.5849,Y 11.4939,Z 59,A -3.1251,B 0.0015,C 0.0015,E1 0.1612,E2 -629.3532} C_DIS
LIN {X -9.2197,Y 12.6155,Z 59,A -3.0783,B 0.0013,C 0.0017,E1 0.161,E2 -629.3026} C_DIS
LIN {X -7.8977,Y 13.4828,Z 59,A -3.0319,B 0.0011,C 0.0018,E1 0.1609,E2 -629.2636} C_DIS
LIN {X -7.164,Y 13.8857,Z 59,A -3.0123,B 0.0011,C 0.0018,E1 0.1607,E2 -629.2391} C_DIS
LIN {X -5.2875,Y 14.7037,Z 59,A -2.9425,B 0.0008,C 0.002,E1 0.1605,E2 -629.2045} C_DIS
LIN {X -3.6535,Y 15.1925,Z 59,A -2.888,B 0.0005,C 0.002,E1 0.1602,E2 -629.1774} C_DIS
LIN {X -1.7486,Y 15.5274,Z 59,A -2.8158,B 0.0003,C 0.0021,E1 0.16,E2 -629.1639} C_DIS
LIN {X -0.179,Y 15.6246,Z 59,A -2.7569,B 0.0001,C 0.0021,E1 0.1598,E2 -629.1596} C_DIS
LIN {X 1.1424,Y 15.5838,Z 59,A -2.7066,B -0.0001,C 0.0021,E1 0.1596,E2 -629.1619} C_DIS
LIN {X 2.3012,Y 15.455,Z 59,A -2.6618,B -0.0003,C 0.0021,E1 0.1594,E2 -629.1683} C_DIS
LIN {X 3.5239,Y 15.2229,Z 59,A -2.6132,B -0.0004,C 0.0021,E1 0.1593,E2 -629.1805} C_DIS
LIN {X 5.0637,Y 14.7822,Z 59,A -2.5501,B -0.0007,C 0.0021,E1 0.1591,E2 -629.2041} C_DIS
LIN {X 6.5031,Y 14.2081,Z 59,A -2.492,B -0.0009,C 0.002,E1 0.1589,E2 -629.2321} C_DIS
LIN {X 7.8292,Y 13.5222,Z 59,A -2.432,B -0.0011,C 0.0019,E1 0.1587,E2 -629.2711} C_DIS
LIN {X 9.1778,Y 12.6461,Z 59,A -2.3777,B -0.0012,C 0.0018,E1 0.1585,E2 -629.3117} C_DIS
LIN {X 10.2979,Y 11.752,Z 59,A -2.3312,B -0.0014,C 0.0016,E1 0.1584,E2 -629.3541} C_DIS
LIN {X 11.1992,Y 10.8968,Z 59,A -2.2869,B -0.0015,C 0.0016,E1 0.1582,E2 -629.4009} C_DIS
LIN {X 12.3235,Y 9.6071,Z 59,A -2.2458,B -0.0016,C 0.0014,E1 0.1581,E2 -629.4549} C_DIS
LIN {X 12.967,Y 8.7186,Z 59,A -2.2045,B -0.0018,C 0.0012,E1 0.158,E2 -629.5102} C_DIS
LIN {X 13.7225,Y 7.4731,Z 59,A -2.1715,B -0.0018,C 0.0011,E1 0.1579,E2 -629.5684} C_DIS
LIN {X 14.2931,Y 6.3137,Z 59,A -2.1417,B -0.0019,C 0.0009,E1 0.1579,E2 -629.6268} C_DIS
LIN {X 14.705,Y 5.2834,Z 59,A -2.1098,B -0.002,C 0.0007,E1 0.1578,E2 -629.6878} C_DIS
LIN {X 15.2555,Y 3.3809,Z 59,A -2.0901,B -0.002,C 0.0005,E1 0.1578,E2 -629.7693} C_DIS
LIN {X 15.4439,Y 2.3644,Z 59,A -2.078,B -0.0021,C 0.0004,E1 0.1577,E2 -629.8185} C_DIS
LIN {X 15.5812,Y 1.1759,Z 59,A -2.0607,B -0.0021,C 0.0002,E1 0.1577,E2 -629.8825} C_DIS
LIN {X 15.6232,Y -0.2674,Z 59,A -2.0421,B -0.0021,C 0,E1 0.1577,E2 -629.9626} C_DIS
LIN {X 15.4544,Y -2.3072,Z 59,A -2.0318,B -0.0021,C -0.0003,E1 0.1577,E2 -630.0682} C_DIS
LIN {X 15.0413,Y -4.2331,Z 59,A -2.0506,B -0.0021,C -0.0005,E1 0.1577,E2 -630.1488} C_DIS
LIN {X 14.57,Y -5.6458,Z 59,A -2.0572,B -0.0021,C -0.0007,E1 0.1578,E2 -630.2215} C_DIS
LIN {X 14.0561,Y -6.825,Z 59,A -2.0656,B -0.0019,C -0.0009,E1 0.1578,E2 -630.2838} C_DIS
LIN {X 13.395,Y -8.0458,Z 59,A -2.0843,B -0.0019,C -0.0011,E1 0.158,E2 -630.343} C_DIS
LIN {X 12.4386,Y -9.4573,Z 59,A -2.1163,B -0.0017,C -0.0013,E1 0.1581,E2 -630.4079} C_DIS
LIN {X 11.3276,Y -10.7623,Z 59,A -2.143,B -0.0016,C -0.0015,E1 0.1583,E2 -630.4792} C_DIS
LIN {X 9.8955,Y -12.0921,Z 59,A -2.1883,B -0.0014,C -0.0017,E1 0.1585,E2 -630.5444} C_DIS
LIN {X 8.3995,Y -13.176,Z 59,A -2.2509,B -0.0012,C -0.0017,E1 0.1587,E2 -630.5835} C_DIS
LIN {X 7.6402,Y -13.6303,Z 59,A -2.2732,B -0.0011,C -0.0018,E1 0.1587,E2 -630.6088} C_DIS
LIN {X 6.5262,Y -14.1951,Z 59,A -2.3133,B -0.0009,C -0.0019,E1 0.1589,E2 -630.6337} C_DIS
LIN {X 5.5262,Y -14.6157,Z 59,A -2.3457,B -0.0008,C -0.0019,E1 0.1591,E2 -630.6559} C_DIS
LIN {X 4.1982,Y -15.0508,Z 59,A -2.3961,B -0.0006,C -0.002,E1 0.1592,E2 -630.6724} C_DIS
LIN {X 3.2049,Y -15.2935,Z 59,A -2.4307,B -0.0005,C -0.002,E1 0.1594,E2 -630.6843} C_DIS
LIN {X 2.0981,Y -15.4837,Z 59,A -2.471,B -0.0003,C -0.0021,E1 0.1596,E2 -630.6923} C_DIS
LIN {X 0.6577,Y -15.6113,Z 59,A -2.5244,B -0.0001,C -0.0021,E1 0.1598,E2 -630.6963} C_DIS
LIN {X 0.6577,Y -15.6113,Z 59,A -2.5244,B -0.0001,C -0.0021,E1 0.1598,E2 -630.6963} C_DIS
Enddeposition()
LIN {X -0.05,Y -14.6387,Z 59,A -2.5074,B -0.0001,C -0.0021,E1 0.1598,E2 -630.6963} C_DIS
Startdeposition()
$VEL.CP = VEL_PRINT
LIN {X 1.6236,Y -14.5545,Z 59,A -2.4501,B -0.0004,C -0.0021,E1 0.1595,E2 -630.6895} C_DIS
LIN {X 2.9056,Y -14.3536,Z 59,A -2.4044,B -0.0005,C -0.0021,E1 0.1594,E2 -630.6802} C_DIS
LIN {X 3.9248,Y -14.109,Z 59,A -2.3723,B -0.0007,C -0.0021,E1 0.1592,E2 -630.6647} C_DIS
LIN {X 4.8139,Y -13.8311,Z 59,A -2.3435,B -0.0008,C -0.002,E1 0.1591,E2 -630.6493} C_DIS
LIN {X 6.1192,Y -13.3052,Z 59,A -2.3027,B -0.001,C -0.0019,E1 0.1589,E2 -630.6198} C_DIS
LIN {X 7.4697,Y -12.5965,Z 59,A -2.2582,B -0.0012,C -0.0018,E1 0.1587,E2 -630.5842} C_DIS
LIN {X 8.38,Y -12.0102,Z 59,A -2.2309,B -0.0013,C -0.0017,E1 0.1585,E2 -630.5528} C_DIS
LIN {X 9.3891,Y -11.239,Z 59,A -2.2044,B -0.0015,C -0.0016,E1 0.1584,E2 -630.5087} C_DIS
LIN {X 10.4555,Y -10.2545,Z 59,A -2.1764,B -0.0016,C -0.0014,E1 0.1582,E2 -630.4546} C_DIS
LIN {X 11.6094,Y -8.9269,Z 59,A -2.142,B -0.0018,C -0.0012,E1 0.1581,E2 -630.3885} C_DIS
LIN {X 12.3143,Y -7.9265,Z 59,A -2.1307,B -0.0018,C -0.001,E1 0.158,E2 -630.3301} C_DIS
LIN {X 12.9777,Y -6.7858,Z 59,A -2.1102,B -0.0019,C -0.0009,E1 0.1579,E2 -630.2763} C_DIS
LIN {X 13.6901,Y -5.2009,Z 59,A -2.1119,B -0.002,C -0.0006,E1 0.1578,E2 -630.1786} C_DIS
LIN {X 14.1492,Y -3.7775,Z 59,A -2.105,B -0.002,C -0.0004,E1 0.1578,E2 -630.1063} C_DIS
LIN {X 14.4375,Y -2.4548,Z 59,A -2.0997,B -0.0021,C -0.0002,E1 0.1577,E2 -630.0431} C_DIS
LIN {X 14.5779,Y -1.3941,Z 59,A -2.1064,B -0.0021,C -0.0001,E1 0.1577,E2 -629.9849} C_DIS
LIN {X 14.6448,Y -0.1294,Z 59,A -2.116,B -0.0021,C 0.0001,E1 0.1577,E2 -629.9177} C_DIS
LIN {X 14.6074,Y 1.047,Z 59,A -2.1352,B -0.0021,C 0.0003,E1 0.1577,E2 -629.8486} C_DIS
LIN {X 14.3952,Y 2.6914,Z 59,A -2.1495,B -0.0021,C 0.0005,E1 0.1577,E2 -629.7707} C_DIS
LIN {X 14.0713,Y 4.058,Z 59,A -2.1859,B -0.0021,C 0.0007,E1 0.1577,E2 -629.6871} C_DIS
LIN {X 13.5427,Y 5.5734,Z 59,A -2.2063,B -0.0019,C 0.0009,E1 0.1578,E2 -629.621} C_DIS
LIN {X 12.8891,Y 6.9526,Z 59,A -2.2529,B -0.0019,C 0.0011,E1 0.1579,E2 -629.5394} C_DIS
LIN {X 12.1434,Y 8.1857,Z 59,A -2.2878,B -0.0017,C 0.0013,E1 0.1581,E2 -629.4795} C_DIS
LIN {X 11.3699,Y 9.2262,Z 59,A -2.3222,B -0.0016,C 0.0014,E1 0.1581,E2 -629.4296} C_DIS
LIN {X 10.6537,Y 10.0483,Z 59,A -2.3604,B -0.0015,C 0.0016,E1 0.1583,E2 -629.3831} C_DIS
LIN {X 9.6424,Y 11.0224,Z 59,A -2.4076,B -0.0013,C 0.0017,E1 0.1584,E2 -629.3324} C_DIS
LIN {X 8.7365,Y 11.7535,Z 59,A -2.4451,B -0.0012,C 0.0017,E1 0.1586,E2 -629.298} C_DIS
LIN {X 7.9713,Y 12.2855,Z 59,A -2.4785,B -0.001,C 0.0019,E1 0.1586,E2 -629.2709} C_DIS
LIN {X 6.9333,Y 12.8996,Z 59,A -2.5225,B -0.0009,C 0.0019,E1 0.1588,E2 -629.24} C_DIS
LIN {X 5.5237,Y 13.5631,Z 59,A -2.5801,B -0.0007,C 0.002,E1 0.159,E2 -629.2075} C_DIS
LIN {X 4.3787,Y 13.9745,Z 59,A -2.6268,B -0.0005,C 0.002,E1 0.1592,E2 -629.1866} C_DIS
LIN {X 2.6861,Y 14.3964,Z 59,A -2.6895,B -0.0003,C 0.0021,E1 0.1594,E2 -629.17} C_DIS
LIN {X 1.6131,Y 14.5535,Z 59,A -2.73,B -0.0001,C 0.0021,E1 0.1596,E2 -629.1634} C_DIS
LIN {X -0.3119,Y 14.6413,Z 59,A -2.7987,B 0.0002,C 0.0021,E1 0.16,E2 -629.1636} C_DIS
LIN {X -1.9395,Y 14.5158,Z 59,A -2.8533,B 0.0005,C 0.0021,E1 0.1602,E2 -629.1753} C_DIS
LIN {X -4.5332,Y 13.9253,Z 59,A -2.9444,B 0.0008,C 0.002,E1 0.1605,E2 -629.2063} C_DIS
LIN {X -6.0311,Y 13.345,Z 59,A -2.9851,B 0.001,C 0.0019,E1 0.1608,E2 -629.2458} C_DIS
LIN {X -7.531,Y 12.56,Z 59,A -3.0336,B 0.0012,C 0.0017,E1 0.1609,E2 -629.286} C_DIS
LIN {X -8.6144,Y 11.8433,Z 59,A -3.0666,B 0.0014,C 0.0017,E1 0.1611,E2 -629.3231} C_DIS
LIN {X -9.6606,Y 11.0064,Z 59,A -3.0913,B 0.0015,C 0.0015,E1 0.1613,E2 -629.372} C_DIS
LIN {X -10.8985,Y 9.7823,Z 59,A -3.1255,B 0.0017,C 0.0013,E1 0.1614,E2 -629.4346} C_DIS
LIN {X -11.647,Y 8.8772,Z 59,A -3.1422,B 0.0017,C 0.0012,E1 0.1615,E2 -629.4831} C_DIS
LIN {X -12.4111,Y 7.774,Z 59,A -3.1555,B 0.0019,C 0.001,E1 0.1616,E2 -629.5439} C_DIS
LIN {X -13.2305,Y 6.2783,Z 59,A -3.1648,B 0.002,C 0.0007,E1 0.1618,E2 -629.6267} C_DIS
LIN {X -13.8435,Y 4.7779,Z 59,A -3.1743,B 0.002,C 0.0005,E1 0.1618,E2 -629.7022} C_DIS
LIN {X -14.239,Y 3.4237,Z 59,A -3.177,B 0.0021,C 0.0003,E1 0.1618,E2 -629.7704} C_DIS
LIN {X -14.5142,Y 1.9516,Z 59,A -3.1677,B 0.0021,C 0.0001,E1 0.1619,E2 -629.851} C_DIS
LIN {X -14.6397,Y 0.3849,Z 59,A -3.158,B 0.0021,C -0.0001,E1 0.1619,E2 -629.9305} C_DIS
LIN {X -14.6092,Y -1.0206,Z 59,A -3.1451,B 0.0021,C -0.0003,E1 0.1619,E2 -630.0011} C_DIS
LIN {X -14.451,Y -2.3588,Z 59,A -3.1334,B 0.0021,C -0.0005,E1 0.1619,E2 -630.0631} C_DIS
LIN {X -14.2389,Y -3.4241,Z 59,A -3.1114,B 0.0021,C -0.0007,E1 0.1619,E2 -630.1221} C_DIS
LIN {X -13.9175,Y -4.5559,Z 59,A -3.0913,B 0.002,C -0.0008,E1 0.1619,E2 -630.1781} C_DIS
LIN {X -13.4819,Y -5.7158,Z 59,A -3.0702,B 0.002,C -0.001,E1 0.1618,E2 -630.2322} C_DIS
LIN {X -12.8899,Y -6.9513,Z 59,A -3.0234,B 0.0018,C -0.0012,E1 0.1616,E2 -630.3096} C_DIS
LIN {X -12.0201,Y -8.3657,Z 59,A -2.9806,B 0.0017,C -0.0014,E1 0.1616,E2 -630.3808} C_DIS
LIN {X -11.1655,Y -9.4764,Z 59,A -2.9448,B 0.0015,C -0.0014,E1 0.1614,E2 -630.4328} C_DIS
LIN {X -10.3831,Y -10.3278,Z 59,A -2.9058,B 0.0014,C -0.0016,E1 0.1613,E2 -630.4799} C_DIS
LIN {X -9.4357,Y -11.1999,Z 59,A -2.8656,B 0.0013,C -0.0017,E1 0.1611,E2 -630.5231} C_DIS
LIN {X -8.3339,Y -12.0422,Z 59,A -2.8218,B 0.0011,C -0.0018,E1 0.161,E2 -630.5632} C_DIS
LIN {X -7.4455,Y -12.6105,Z 59,A -2.7852,B 0.001,C -0.0019,E1 0.1609,E2 -630.5921} C_DIS
LIN {X -6.2944,Y -13.2214,Z 59,A -2.7402,B 0.0008,C -0.0019,E1 0.1607,E2 -630.622} C_DIS
LIN {X -4.9325,Y -13.789,Z 59,A -2.6819,B 0.0006,C -0.0021,E1 0.1605,E2 -630.6557} C_DIS
LIN {X -3.3202,Y -14.2635,Z 59,A -2.6233,B 0.0003,C -0.0021,E1 0.1602,E2 -630.6768} C_DIS
LIN {X -2.1945,Y -14.4795,Z 59,A -2.5813,B 0.0002,C -0.0021,E1 0.1601,E2 -630.6876} C_DIS
LIN {X -0.9802,Y -14.612,Z 59,A -2.5369,B 0,C -0.0021,E1 0.1599,E2 -630.694} C_DIS
LIN {X -0.05,Y -14.6387,Z 59,A -2.5035,B -0.0001,C -0.0021,E1 0.1598,E2 -630.695} C_DIS
Enddeposition()
LIN {X -0.05,Y -14.6387,Z 59,A -2.5035,B -0.0001,C -0.0021,E1 0.1598,E2 -630.695} C_DIS
Startdeposition()
$VEL.CP = VEL_PRINT
LIN {X -0.4777,Y -13.6553,Z 59,A -2.4701,B 0,C -0.0021,E1 0.1599,E2 -630.7009} C_DIS
LIN {X -2.6661,Y -13.4009,Z 59,A -2.561,B 0.0004,C -0.0021,E1 0.1603,E2 -630.6778} C_DIS
LIN {X -4.4147,Y -12.9311,Z 59,A -2.6292,B 0.0007,C -0.0021,E1 0.1605,E2 -630.6522} C_DIS
LIN {X -5.5879,Y -12.4691,Z 59,A -2.6795,B 0.0008,C -0.002,E1 0.1607,E2 -630.6243} C_DIS
LIN {X -6.8797,Y -11.8055,Z 59,A -2.7423,B 0.0011,C -0.0019,E1 0.1609,E2 -630.5795} C_DIS
LIN {X -8.2723,Y -10.8755,Z 59,A -2.8069,B 0.0013,C -0.0017,E1 0.1612,E2 -630.5253} C_DIS
LIN {X -9.6206,Y -9.7031,Z 59,A -2.8695,B 0.0015,C -0.0016,E1 0.1614,E2 -630.4613} C_DIS
LIN {X -10.51,Y -8.7318,Z 59,A -2.9156,B 0.0016,C -0.0014,E1 0.1614,E2 -630.406} C_DIS
LIN {X -11.1709,Y -7.8691,Z 59,A -2.9542,B 0.0017,C -0.0013,E1 0.1616,E2 -630.3547} C_DIS
LIN {X -11.6762,Y -7.0974,Z 59,A -2.9846,B 0.0018,C -0.0012,E1 0.1616,E2 -630.3099} C_DIS
LIN {X -12.4452,Y -5.6409,Z 59,A -3.0381,B 0.0019,C -0.0009,E1 0.1618,E2 -630.2227} C_DIS
LIN {X -13.0251,Y -4.1279,Z 59,A -3.0706,B 0.002,C -0.0007,E1 0.1618,E2 -630.1474} C_DIS
LIN {X -13.3987,Y -2.679,Z 59,A -3.1222,B 0.0021,C -0.0005,E1 0.1619,E2 -630.0488} C_DIS
LIN {X -13.5932,Y -1.3888,Z 59,A -3.154,B 0.0021,C -0.0002,E1 0.1619,E2 -629.97} C_DIS
LIN {X -13.6023,Y 1.2977,Z 59,A -3.172,B 0.0021,C 0.0001,E1 0.1619,E2 -629.84} C_DIS
LIN {X -13.3065,Y 3.1055,Z 59,A -3.2013,B 0.0021,C 0.0005,E1 0.1619,E2 -629.7247} C_DIS
LIN {X -12.8274,Y 4.707,Z 59,A -3.1983,B 0.0021,C 0.0007,E1 0.1619,E2 -629.6433} C_DIS
LIN {X -12.095,Y 6.3563,Z 59,A -3.1793,B 0.002,C 0.0009,E1 0.1617,E2 -629.5667} C_DIS
LIN {X -11.4974,Y 7.383,Z 59,A -3.1932,B 0.0018,C 0.0011,E1 0.1616,E2 -629.4883} C_DIS
LIN {X -10.1925,Y 9.1005,Z 59,A -3.166,B 0.0016,C 0.0014,E1 0.1614,E2 -629.3959} C_DIS
LIN {X -8.3505,Y 10.8154,Z 59,A -3.1232,B 0.0013,C 0.0017,E1 0.161,E2 -629.299} C_DIS
LIN {X -6.2411,Y 12.1552,Z 59,A -3.0498,B 0.001,C 0.0019,E1 0.1608,E2 -629.2378} C_DIS
LIN {X -5.1579,Y 12.6528,Z 59,A -3.0188,B 0.0009,C 0.0019,E1 0.1606,E2 -629.2075} C_DIS
LIN {X -3.7524,Y 13.1384,Z 59,A -2.973,B 0.0006,C 0.0021,E1 0.1603,E2 -629.1805} C_DIS
LIN {X -2.1203,Y 13.4985,Z 59,A -2.9151,B 0.0004,C 0.0021,E1 0.1601,E2 -629.162} C_DIS
LIN {X -0.7867,Y 13.641,Z 59,A -2.8665,B 0.0002,C 0.0021,E1 0.1599,E2 -629.1544} C_DIS
LIN {X 0.7923,Y 13.641,Z 59,A -2.8065,B -0.0001,C 0.0021,E1 0.1596,E2 -629.155} C_DIS
LIN {X 1.8201,Y 13.542,Z 59,A -2.7658,B -0.0002,C 0.0021,E1 0.1595,E2 -629.1611} C_DIS
LIN {X 3.0267,Y 13.3242,Z 59,A -2.7153,B -0.0004,C 0.0021,E1 0.1593,E2 -629.1753} C_DIS
LIN {X 4.5809,Y 12.8731,Z 59,A -2.6502,B -0.0007,C 0.0021,E1 0.159,E2 -629.2007} C_DIS
LIN {X 5.6529,Y 12.4399,Z 59,A -2.6019,B -0.0009,C 0.002,E1 0.1589,E2 -629.2268} C_DIS
LIN {X 6.7684,Y 11.87,Z 59,A -2.5528,B -0.001,C 0.002,E1 0.1587,E2 -629.2581} C_DIS
LIN {X 7.7683,Y 11.2408,Z 59,A -2.5071,B -0.0012,C 0.0018,E1 0.1585,E2 -629.2927} C_DIS
LIN {X 8.6856,Y 10.5484,Z 59,A -2.4614,B -0.0013,C 0.0018,E1 0.1584,E2 -629.3333} C_DIS
LIN {X 9.6828,Y 9.6412,Z 59,A -2.4057,B -0.0015,C 0.0015,E1 0.1582,E2 -629.3901} C_DIS
LIN {X 10.6579,Y 8.5507,Z 59,A -2.3536,B -0.0017,C 0.0014,E1 0.1581,E2 -629.4522} C_DIS
LIN {X 11.5187,Y 7.3502,Z 59,A -2.3048,B -0.0017,C 0.0012,E1 0.158,E2 -629.5202} C_DIS
LIN {X 12.1211,Y 6.3062,Z 59,A -2.271,B -0.0019,C 0.001,E1 0.1579,E2 -629.5763} C_DIS
LIN {X 12.7835,Y 4.8245,Z 59,A -2.2122,B -0.002,C 0.0008,E1 0.1578,E2 -629.6743} C_DIS
LIN {X 13.3257,Y 3.0218,Z 59,A -2.1809,B -0.002,C 0.0005,E1 0.1577,E2 -629.7633} C_DIS
LIN {X 13.5543,Y 1.728,Z 59,A -2.1373,B -0.0021,C 0.0003,E1 0.1577,E2 -629.8546} C_DIS
LIN {X 13.666,Y 0.0086,Z 59,A -2.1171,B -0.0021,C 0,E1 0.1577,E2 -629.9454} C_DIS
LIN {X 13.5661,Y -1.6327,Z 59,A -2.0879,B -0.0021,C -0.0003,E1 0.1577,E2 -630.05} C_DIS
LIN {X 13.203,Y -3.5192,Z 59,A -2.0828,B -0.0021,C -0.0005,E1 0.1577,E2 -630.1509} C_DIS
LIN {X 12.7103,Y -5.0144,Z 59,A -2.0918,B -0.0021,C -0.0007,E1 0.1578,E2 -630.2254} C_DIS
LIN {X 12.2487,Y -6.0559,Z 59,A -2.0949,B -0.002,C -0.0009,E1 0.1578,E2 -630.2849} C_DIS
LIN {X 11.6855,Y -7.0821,Z 59,A -2.0949,B -0.0019,C -0.0011,E1 0.158,E2 -630.3507} C_DIS
LIN {X 10.9056,Y -8.2325,Z 59,A -2.1071,B -0.0017,C -0.0013,E1 0.1581,E2 -630.4176} C_DIS
LIN {X 9.8233,Y -9.4972,Z 59,A -2.1408,B -0.0016,C -0.0015,E1 0.1583,E2 -630.4788} C_DIS
LIN {X 9.0868,Y -10.2023,Z 59,A -2.1594,B -0.0015,C -0.0015,E1 0.1583,E2 -630.5179} C_DIS
LIN {X 7.9483,Y -11.1144,Z 59,A -2.1827,B -0.0013,C -0.0017,E1 0.1586,E2 -630.5762} C_DIS
LIN {X 6.7649,Y -11.8719,Z 59,A -2.2171,B -0.0011,C -0.0019,E1 0.1588,E2 -630.618} C_DIS
LIN {X 4.841,Y -12.7777,Z 59,A -2.2759,B -0.0007,C -0.002,E1 0.1591,E2 -630.6685} C_DIS
LIN {X 2.0961,Y -13.5023,Z 59,A -2.3796,B -0.0004,C -0.0021,E1 0.1595,E2 -630.6956} C_DIS
LIN {X 0.6562,Y -13.6484,Z 59,A -2.4312,B -0.0001,C -0.0021,E1 0.1598,E2 -630.7023} C_DIS
LIN {X 0.6562,Y -13.6484,Z 59,A -2.4312,B -0.0001,C -0.0021,E1 0.1598,E2 -630.7023} C_DIS
Enddeposition()
LIN {X -0.039,Y -12.6826,Z 59,A -2.4149,B -0.0001,C -0.0021,E1 0.1598,E2 -630.7015} C_DIS
Startdeposition()
$VEL.CP = VEL_PRINT
LIN {X 1.2333,Y -12.6231,Z 59,A -2.3713,B -0.0003,C -0.0021,E1 0.1596,E2 -630.6965} C_DIS
LIN {X 3.071,Y -12.3059,Z 59,A -2.3161,B -0.0007,C -0.0021,E1 0.1592,E2 -630.6714} C_DIS
LIN {X 4.5632,Y -11.834,Z 59,A -2.2672,B -0.0009,C -0.002,E1 0.159,E2 -630.6458} C_DIS
LIN {X 5.7773,Y -11.291,Z 59,A -2.2374,B -0.0011,C -0.0018,E1 0.1588,E2 -630.6077} C_DIS
LIN {X 7.2328,Y -10.4181,Z 59,A -2.1995,B -0.0013,C -0.0017,E1 0.1585,E2 -630.5545} C_DIS
LIN {X 8.4343,Y -9.4726,Z 59,A -2.1634,B -0.0015,C -0.0015,E1 0.1584,E2 -630.5054} C_DIS
LIN {X 9.4513,Y -8.458,Z 59,A -2.167,B -0.0017,C -0.0013,E1 0.1581,E2 -630.42} C_DIS
LIN {X 10.2856,Y -7.4211,Z 59,A -2.1507,B -0.0018,C -0.0011,E1 0.1581,E2 -630.3603} C_DIS
LIN {X 11.2321,Y -5.8906,Z 59,A -2.1281,B -0.002,C -0.0009,E1 0.1579,E2 -630.2812} C_DIS
LIN {X 11.6281,Y -5.0648,Z 59,A -2.1534,B -0.002,C -0.0007,E1 0.1578,E2 -630.2049} C_DIS
LIN {X 12.3708,Y -2.7972,Z 59,A -2.1764,B -0.0021,C -0.0003,E1 0.1577,E2 -630.0551} C_DIS
LIN {X 12.6842,Y 0.0625,Z 59,A -2.1837,B -0.0021,C 0.0001,E1 0.1577,E2 -629.9118} C_DIS
LIN {X 12.6842,Y 0.0625,Z 59,A -2.1848,B -0.0021,C 0.0001,E1 0.1577,E2 -629.9106} C_DIS
LIN {X 12.568,Y 1.703,Z 59,A -2.2412,B -0.0021,C 0.0005,E1 0.1577,E2 -629.7871} C_DIS
LIN {X 12.2091,Y 3.4351,Z 59,A -2.2715,B -0.0021,C 0.0007,E1 0.1577,E2 -629.6952} C_DIS
LIN {X 11.812,Y 4.6196,Z 59,A -2.305,B -0.002,C 0.0009,E1 0.1578,E2 -629.6253} C_DIS
LIN {X 11.2696,Y 5.8187,Z 59,A -2.3533,B -0.0018,C 0.0011,E1 0.1579,E2 -629.5456} C_DIS
LIN {X 10.7371,Y 6.7514,Z 59,A -2.3808,B -0.0018,C 0.0013,E1 0.1579,E2 -629.498} C_DIS
LIN {X 9.9474,Y 7.8686,Z 59,A -2.4343,B -0.0016,C 0.0015,E1 0.1581,E2 -629.4263} C_DIS
LIN {X 9.2569,Y 8.6704,Z 59,A -2.4722,B -0.0015,C 0.0015,E1 0.1583,E2 -629.3801} C_DIS
LIN {X 8.2594,Y 9.6254,Z 59,A -2.5256,B -0.0013,C 0.0017,E1 0.1584,E2 -629.3235} C_DIS
LIN {X 7.2338,Y 10.4181,Z 59,A -2.5736,B -0.0011,C 0.0018,E1 0.1586,E2 -629.2805} C_DIS
LIN {X 5.7939,Y 11.2825,Z 59,A -2.6477,B -0.0008,C 0.002,E1 0.1589,E2 -629.224} C_DIS
LIN {X 4.6765,Y 11.7896,Z 59,A -2.6992,B -0.0006,C 0.002,E1 0.1591,E2 -629.1932} C_DIS
LIN {X 2.5975,Y 12.4144,Z 59,A -2.7791,B -0.0003,C 0.0021,E1 0.1594,E2 -629.1653} C_DIS
LIN {X 0.916,Y 12.6502,Z 59,A -2.8415,B 0,C 0.0021,E1 0.1597,E2 -629.1564} C_DIS
LIN {X -1.0963,Y 12.6358,Z 59,A -2.9101,B 0.0004,C 0.0021,E1 0.1601,E2 -629.1641} C_DIS
LIN {X -2.9545,Y 12.3343,Z 59,A -2.9668,B 0.0007,C 0.0021,E1 0.1604,E2 -629.1897} C_DIS
LIN {X -5.364,Y 11.4932,Z 59,A -3.0401,B 0.0011,C 0.0019,E1 0.1608,E2 -629.2417} C_DIS
LIN {X -6.862,Y 10.6665,Z 59,A -3.0708,B 0.0013,C 0.0017,E1 0.161,E2 -629.3012} C_DIS
LIN {X -8.1498,Y 9.7184,Z 59,A -3.1032,B 0.0015,C 0.0015,E1 0.1612,E2 -629.3562} C_DIS
LIN {X -9.0706,Y 8.8652,Z 59,A -3.1207,B 0.0017,C 0.0014,E1 0.1614,E2 -629.4083} C_DIS
LIN {X -9.8214,Y 8.0253,Z 59,A -3.1337,B 0.0017,C 0.0012,E1 0.1614,E2 -629.4581} C_DIS
LIN {X -10.5859,Y 6.9859,Z 59,A -3.1356,B 0.0019,C 0.001,E1 0.1616,E2 -629.5276} C_DIS
LIN {X -11.4267,Y 5.5028,Z 59,A -3.1254,B 0.002,C 0.0007,E1 0.1618,E2 -629.6302} C_DIS
LIN {X -12.0503,Y 3.9565,Z 59,A -3.1134,B 0.0021,C 0.0005,E1 0.1618,E2 -629.7294} C_DIS
LIN {X -12.5976,Y 1.4715,Z 59,A -3.1127,B 0.0021,C 0.0001,E1 0.1619,E2 -629.854} C_DIS
LIN {X -12.6824,Y 0.1592,Z 59,A -3.0761,B 0.0021,C -0.0002,E1 0.1619,E2 -629.9483} C_DIS
LIN {X -12.6073,Y -1.3856,Z 59,A -3.0552,B 0.0021,C -0.0004,E1 0.1619,E2 -630.0311} C_DIS
LIN {X -12.4188,Y -2.5734,Z 59,A -3.0259,B 0.0021,C -0.0006,E1 0.1619,E2 -630.1034} C_DIS
LIN {X -12.0986,Y -3.8064,Z 59,A -2.9962,B 0.0021,C -0.0008,E1 0.1619,E2 -630.1733} C_DIS
LIN {X -11.4974,Y -5.3549,Z 59,A -2.9405,B 0.0019,C -0.0011,E1 0.1617,E2 -630.2724} C_DIS
LIN {X -11.0659,Y -6.1976,Z 59,A -2.9124,B 0.0018,C -0.0011,E1 0.1617,E2 -630.3206} C_DIS
LIN {X -10.4751,Y -7.1511,Z 59,A -2.876,B 0.0017,C -0.0013,E1 0.1615,E2 -630.3759} C_DIS
LIN {X -9.8572,Y -7.9812,Z 59,A -2.8364,B 0.0016,C -0.0015,E1 0.1615,E2 -630.4284} C_DIS
LIN {X -8.916,Y -9.0205,Z 59,A -2.7855,B 0.0014,C -0.0016,E1 0.1613,E2 -630.4896} C_DIS
LIN {X -7.9456,Y -9.8857,Z 59,A -2.7433,B 0.0012,C -0.0018,E1 0.1611,E2 -630.5336} C_DIS
LIN {X -7.031,Y -10.556,Z 59,A -2.6976,B 0.0011,C -0.0018,E1 0.161,E2 -630.575} C_DIS
LIN {X -6.2175,Y -11.0548,Z 59,A -2.6598,B 0.0009,C -0.0019,E1 0.1608,E2 -630.605} C_DIS
LIN {X -5.0507,Y -11.6343,Z 59,A -2.6035,B 0.0007,C -0.002,E1 0.1606,E2 -630.6442} C_DIS
LIN {X -3.7017,Y -12.131,Z 59,A -2.5498,B 0.0005,C -0.0021,E1 0.1604,E2 -630.6707} C_DIS
LIN {X -2.3992,Y -12.4537,Z 59,A -2.4996,B 0.0003,C -0.0021,E1 0.1602,E2 -630.6878} C_DIS
LIN {X -1.1025,Y -12.6353,Z 59,A -2.45,B 0,C -0.0021,E1 0.1599,E2 -630.6986} C_DIS
LIN {X -0.039,Y -12.6826,Z 59,A -2.4122,B 0,C -0.0021,E1 0.1599,E2 -630.7002} C_DIS
Enddeposition()
LIN {X -0.039,Y -12.6826,Z 59,A -2.4122,B 0,C -0.0021,E1 0.1599,E2 -630.7002} C_DIS
Startdeposition()
$VEL.CP = VEL_PRINT
LIN {X -0.7341,Y -11.6794,Z 59,A -2.3932,B 0,C -0.0021,E1 0.1599,E2 -630.7005} C_DIS
LIN {X -2.4097,Y -11.4515,Z 59,A -2.4686,B 0.0005,C -0.0021,E1 0.1603,E2 -630.6756} C_DIS
LIN {X -4.4156,Y -10.8374,Z 59,A -2.5588,B 0.0008,C -0.0021,E1 0.1607,E2 -630.6312} C_DIS
LIN {X -5.4646,Y -10.3482,Z 59,A -2.6094,B 0.001,C -0.0019,E1 0.1609,E2 -630.5974} C_DIS
LIN {X -6.7483,Y -9.561,Z 59,A -2.6751,B 0.0012,C -0.0018,E1 0.1611,E2 -630.5442} C_DIS
LIN {X -7.6771,Y -8.8323,Z 59,A -2.7292,B 0.0014,C -0.0017,E1 0.1613,E2 -630.4924} C_DIS
LIN {X -8.713,Y -7.8123,Z 59,A -2.7952,B 0.0016,C -0.0015,E1 0.1615,E2 -630.4204} C_DIS
LIN {X -9.7212,Y -6.5152,Z 59,A -2.8592,B 0.0018,C -0.0012,E1 0.1616,E2 -630.3377} C_DIS
LIN {X -10.2344,Y -5.6751,Z 59,A -2.9039,B 0.0018,C -0.0011,E1 0.1617,E2 -630.2761} C_DIS
LIN {X -11.0013,Y -3.99,Z 59,A -2.9706,B 0.002,C -0.0008,E1 0.1619,E2 -630.1661} C_DIS
LIN {X -11.4304,Y -2.5079,Z 59,A -3.0163,B 0.002,C -0.0005,E1 0.1619,E2 -630.0736} C_DIS
LIN {X -11.6381,Y -1.226,Z 59,A -3.0552,B 0.0021,C -0.0003,E1 0.1619,E2 -629.9885} C_DIS
LIN {X -11.7007,Y 0.2034,Z 59,A -3.0965,B 0.0021,C 0,E1 0.1619,E2 -629.8897} C_DIS
LIN {X -11.5861,Y 1.6465,Z 59,A -3.1237,B 0.0021,C 0.0003,E1 0.1619,E2 -629.7981} C_DIS
LIN {X -11.2586,Y 3.1919,Z 59,A -3.1449,B 0.0021,C 0.0005,E1 0.1619,E2 -629.7004} C_DIS
LIN {X -10.8717,Y 4.33,Z 59,A -3.1472,B 0.0021,C 0.0007,E1 0.1618,E2 -629.6364} C_DIS
LIN {X -10.4827,Y 5.2013,Z 59,A -3.1584,B 0.002,C 0.0009,E1 0.1618,E2 -629.5747} C_DIS
LIN {X -9.6776,Y 6.5794,Z 59,A -3.1791,B 0.0018,C 0.0012,E1 0.1615,E2 -629.4672} C_DIS
LIN {X -8.6388,Y 7.894,Z 59,A -3.17,B 0.0016,C 0.0015,E1 0.1613,E2 -629.3831} C_DIS
LIN {X -6.9711,Y 9.3996,Z 59,A -3.1308,B 0.0013,C 0.0017,E1 0.161,E2 -629.2976} C_DIS
LIN {X -5.5784,Y 10.287,Z 59,A -3.0982,B 0.0011,C 0.0019,E1 0.1608,E2 -629.2413} C_DIS
LIN {X -4.7792,Y 10.6819,Z 59,A -3.0837,B 0.0009,C 0.0019,E1 0.1606,E2 -629.2095} C_DIS
LIN {X -2.4871,Y 11.4349,Z 59,A -3.0049,B 0.0005,C 0.0021,E1 0.1602,E2 -629.1709} C_DIS
LIN {X -1.0832,Y 11.6522,Z 59,A -2.9595,B 0.0002,C 0.0021,E1 0.1599,E2 -629.1546} C_DIS
LIN {X 0.664,Y 11.6836,Z 59,A -2.8924,B -0.0001,C 0.0021,E1 0.1596,E2 -629.1546} C_DIS
LIN {X 1.9713,Y 11.5326,Z 59,A -2.842,B -0.0003,C 0.0021,E1 0.1594,E2 -629.1621} C_DIS
LIN {X 2.7901,Y 11.3651,Z 59,A -2.802,B -0.0005,C 0.0021,E1 0.1592,E2 -629.1783} C_DIS
LIN {X 4.1388,Y 10.9461,Z 59,A -2.7427,B -0.0007,C 0.0021,E1 0.159,E2 -629.2044} C_DIS
LIN {X 5.3787,Y 10.393,Z 59,A -2.6786,B -0.001,C 0.0019,E1 0.1588,E2 -629.2451} C_DIS
LIN {X 6.5034,Y 9.7292,Z 59,A -2.6172,B -0.0012,C 0.0019,E1 0.1585,E2 -629.2923} C_DIS
LIN {X 7.6597,Y 8.8472,Z 59,A -2.5605,B -0.0014,C 0.0017,E1 0.1584,E2 -629.343} C_DIS
LIN {X 8.3699,Y 8.1789,Z 59,A -2.5189,B -0.0014,C 0.0016,E1 0.1582,E2 -629.3863} C_DIS
LIN {X 9.0509,Y 7.4181,Z 59,A -2.4568,B -0.0017,C 0.0014,E1 0.1581,E2 -629.4553} C_DIS
LIN {X 9.8227,Y 6.3609,Z 59,A -2.4001,B -0.0018,C 0.0012,E1 0.1579,E2 -629.5284} C_DIS
LIN {X 10.6631,Y 4.8216,Z 59,A -2.3357,B -0.002,C 0.0009,E1 0.1578,E2 -629.6275} C_DIS
LIN {X 11.2296,Y 3.2915,Z 59,A -2.2823,B -0.002,C 0.0006,E1 0.1578,E2 -629.7258} C_DIS
LIN {X 11.5278,Y 2.0139,Z 59,A -2.2395,B -0.0021,C 0.0004,E1 0.1577,E2 -629.8128} C_DIS
LIN {X 11.6855,Y 0.6294,Z 59,A -2.1979,B -0.0021,C 0.0001,E1 0.1577,E2 -629.9087} C_DIS
LIN {X 11.6615,Y -0.9754,Z 59,A -2.1524,B -0.0021,C -0.0002,E1 0.1577,E2 -630.025} C_DIS
LIN {X 11.4375,Y -2.4755,Z 59,A -2.1393,B -0.0021,C -0.0004,E1 0.1577,E2 -630.1117} C_DIS
LIN {X 11.1398,Y -3.5844,Z 59,A -2.1329,B -0.0021,C -0.0006,E1 0.1577,E2 -630.1775} C_DIS
LIN {X 10.8257,Y -4.4444,Z 59,A -2.1172,B -0.0021,C -0.0008,E1 0.1578,E2 -630.2425} C_DIS
LIN {X 10.3,Y -5.5477,Z 59,A -2.1166,B -0.0019,C -0.001,E1 0.1579,E2 -630.3107} C_DIS
LIN {X 9.8567,Y -6.304,Z 59,A -2.1158,B -0.0019,C -0.0011,E1 0.1579,E2 -630.361} C_DIS
LIN {X 9.0761,Y -7.3873,Z 59,A -2.114,B -0.0017,C -0.0014,E1 0.1582,E2 -630.4389} C_DIS
LIN {X 8.2412,Y -8.3086,Z 59,A -2.1277,B -0.0015,C -0.0015,E1 0.1583,E2 -630.496} C_DIS
LIN {X 7.2947,Y -9.1508,Z 59,A -2.1423,B -0.0014,C -0.0017,E1 0.1585,E2 -630.5528} C_DIS
LIN {X 6.2832,Y -9.8728,Z 59,A -2.1673,B -0.0012,C -0.0018,E1 0.1587,E2 -630.5963} C_DIS
LIN {X 5.2582,Y -10.4544,Z 59,A -2.1873,B -0.001,C -0.0019,E1 0.1589,E2 -630.639} C_DIS
LIN {X 3.3098,Y -11.2244,Z 59,A -2.2518,B -0.0006,C -0.0021,E1 0.1592,E2 -630.6786} C_DIS
LIN {X 2.1857,Y -11.4965,Z 59,A -2.2891,B -0.0004,C -0.0021,E1 0.1594,E2 -630.6939} C_DIS
LIN {X 1.0268,Y -11.6573,Z 59,A -2.3302,B -0.0002,C -0.0021,E1 0.1597,E2 -630.7016} C_DIS
LIN {X -0.0599,Y -11.7016,Z 59,A -2.37,B -0.0002,C -0.0021,E1 0.1597,E2 -630.7029} C_DIS
Enddeposition()
LIN {X -0.0599,Y -11.7016,Z 59,A -2.37,B -0.0002,C -0.0021,E1 0.1597,E2 -630.7029} C_DIS
Startdeposition()
$VEL.CP = VEL_PRINT
LIN {X 0.4274,Y -10.7132,Z 59,A -2.3193,B -0.0002,C -0.0021,E1 0.1597,E2 -630.6929} C_DIS
LIN {X 2.2082,Y -10.4918,Z 59,A -2.2601,B -0.0005,C -0.0021,E1 0.1593,E2 -630.6781} C_DIS
LIN {X 3.1035,Y -10.2623,Z 59,A -2.2372,B -0.0007,C -0.0021,E1 0.1591,E2 -630.6585} C_DIS
LIN {X 4.2574,Y -9.84,Z 59,A -2.2137,B -0.001,C -0.0019,E1 0.1589,E2 -630.6217} C_DIS
LIN {X 5.4782,Y -9.2166,Z 59,A -2.1948,B -0.0013,C -0.0017,E1 0.1586,E2 -630.5689} C_DIS
LIN {X 7.1124,Y -8.0232,Z 59,A -2.1717,B -0.0016,C -0.0015,E1 0.1583,E2 -630.4801} C_DIS
LIN {X 8.6328,Y -6.3587,Z 59,A -2.1512,B -0.0018,C -0.0012,E1 0.1581,E2 -630.3722} C_DIS
LIN {X 9.2922,Y -5.3488,Z 59,A -2.156,B -0.0019,C -0.001,E1 0.1579,E2 -630.299} C_DIS
LIN {X 9.7567,Y -4.4449,Z 59,A -2.175,B -0.002,C -0.0007,E1 0.1579,E2 -630.2232} C_DIS
LIN {X 10.2204,Y -3.2406,Z 59,A -2.1809,B -0.002,C -0.0005,E1 0.1577,E2 -630.1477} C_DIS
LIN {X 10.5032,Y -2.1535,Z 59,A -2.2077,B -0.0021,C -0.0003,E1 0.1577,E2 -630.0629} C_DIS
LIN {X 10.6651,Y -1.0983,Z 59,A -2.2275,B -0.0021,C -0.0001,E1 0.1577,E2 -629.9911} C_DIS
LIN {X 10.6732,Y 1.0151,Z 59,A -2.3237,B -0.0021,C 0.0004,E1 0.1577,E2 -629.8024} C_DIS
LIN {X 10.137,Y 3.492,Z 59,A -2.3942,B -0.002,C 0.0009,E1 0.1578,E2 -629.6449} C_DIS
LIN {X 9.7256,Y 4.5131,Z 59,A -2.4296,B -0.0019,C 0.001,E1 0.1578,E2 -629.5809} C_DIS
LIN {X 9.1623,Y 5.5632,Z 59,A -2.4735,B -0.0018,C 0.0012,E1 0.158,E2 -629.513} C_DIS
LIN {X 8.442,Y 6.6099,Z 59,A -2.539,B -0.0016,C 0.0014,E1 0.1582,E2 -629.4296} C_DIS
LIN {X 7.4937,Y 7.6683,Z 59,A -2.6025,B -0.0014,C 0.0016,E1 0.1584,E2 -629.3566} C_DIS
LIN {X 6.4832,Y 8.5397,Z 59,A -2.6646,B -0.0011,C 0.0018,E1 0.1586,E2 -629.2954} C_DIS
LIN {X 5.2253,Y 9.3623,Z 59,A -2.7278,B -0.0009,C 0.0019,E1 0.1588,E2 -629.2447} C_DIS
LIN {X 4.0606,Y 9.9231,Z 59,A -2.7872,B -0.0006,C 0.002,E1 0.1591,E2 -629.2055} C_DIS
LIN {X 2.7324,Y 10.3676,Z 59,A -2.8448,B -0.0004,C 0.0021,E1 0.1593,E2 -629.1791} C_DIS
LIN {X 1.4733,Y 10.6173,Z 59,A -2.8949,B -0.0001,C 0.0021,E1 0.1596,E2 -629.166} C_DIS
LIN {X 0.2862,Y 10.7178,Z 59,A -2.9393,B 0.0001,C 0.0021,E1 0.1598,E2 -629.162} C_DIS
LIN {X -1.1871,Y 10.6558,Z 59,A -2.9867,B 0.0004,C 0.0021,E1 0.1601,E2 -629.1726} C_DIS
LIN {X -2.6741,Y 10.3828,Z 59,A -3.0305,B 0.0007,C 0.0021,E1 0.1604,E2 -629.196} C_DIS
LIN {X -4.0358,Y 9.9328,Z 59,A -3.0678,B 0.0009,C 0.0019,E1 0.1606,E2 -629.2284} C_DIS
LIN {X -5.293,Y 9.3242,Z 59,A -3.0901,B 0.0012,C 0.0018,E1 0.1609,E2 -629.2784} C_DIS
LIN {X -6.2725,Y 8.6956,Z 59,A -3.1088,B 0.0014,C 0.0016,E1 0.1611,E2 -629.3223} C_DIS
LIN {X -7.5695,Y 7.5929,Z 59,A -3.1134,B 0.0016,C 0.0014,E1 0.1614,E2 -629.4117} C_DIS
LIN {X -8.726,Y 6.2291,Z 59,A -3.0998,B 0.0019,C 0.001,E1 0.1616,E2 -629.5247} C_DIS
LIN {X -9.6789,Y 4.612,Z 59,A -3.1017,B 0.002,C 0.0008,E1 0.1618,E2 -629.6253} C_DIS
LIN {X -10.1155,Y 3.5543,Z 59,A -3.0853,B 0.002,C 0.0005,E1 0.1618,E2 -629.7019} C_DIS
LIN {X -10.4476,Y 2.4086,Z 59,A -3.0664,B 0.0021,C 0.0003,E1 0.1618,E2 -629.7807} C_DIS
LIN {X -10.6497,Y 1.2402,Z 59,A -3.0388,B 0.0021,C 0.0001,E1 0.1619,E2 -629.8645} C_DIS
LIN {X -10.7228,Y 0.0274,Z 59,A -3.0123,B 0.0021,C -0.0002,E1 0.1619,E2 -629.9444} C_DIS
LIN {X -10.6799,Y -0.9466,Z 59,A -2.9773,B 0.0021,C -0.0004,E1 0.1619,E2 -630.0186} C_DIS
LIN {X -10.4323,Y -2.4746,Z 59,A -2.925,B 0.0021,C -0.0007,E1 0.1619,E2 -630.126} C_DIS
LIN {X -10.042,Y -3.7564,Z 59,A -2.8799,B 0.0019,C -0.0009,E1 0.1618,E2 -630.2109} C_DIS
LIN {X -9.5068,Y -4.9573,Z 59,A -2.8172,B 0.0019,C -0.0011,E1 0.1616,E2 -630.3049} C_DIS
LIN {X -8.5788,Y -6.4311,Z 59,A -2.7396,B 0.0016,C -0.0014,E1 0.1614,E2 -630.4114} C_DIS
LIN {X -7.3982,Y -7.7605,Z 59,A -2.6706,B 0.0014,C -0.0017,E1 0.1612,E2 -630.4943} C_DIS
LIN {X -6.4795,Y -8.5424,Z 59,A -2.619,B 0.0012,C -0.0017,E1 0.161,E2 -630.5462} C_DIS
LIN {X -5.6017,Y -9.1421,Z 59,A -2.5714,B 0.001,C -0.0019,E1 0.1609,E2 -630.5878} C_DIS
LIN {X -4.6331,Y -9.6672,Z 59,A -2.5253,B 0.0008,C -0.0019,E1 0.1607,E2 -630.6214} C_DIS
LIN {X -3.7836,Y -10.0319,Z 59,A -2.4822,B 0.0006,C -0.002,E1 0.1605,E2 -630.6496} C_DIS
LIN {X -2.6401,Y -10.3915,Z 59,A -2.4332,B 0.0004,C -0.0021,E1 0.1603,E2 -630.6729} C_DIS
LIN {X -1.63,Y -10.597,Z 59,A -2.3919,B 0.0002,C -0.0021,E1 0.1601,E2 -630.6867} C_DIS
LIN {X -0.5613,Y -10.707,Z 59,A -2.3514,B 0,C -0.0021,E1 0.1599,E2 -630.6934} C_DIS
LIN {X -0.5613,Y -10.707,Z 59,A -2.3514,B 0,C -0.0021,E1 0.1599,E2 -630.6934} C_DIS
Enddeposition()
LIN {X -0.0615,Y -9.7408,Z 59,A -2.2896,B 0,C -0.0021,E1 0.1599,E2 -630.6951} C_DIS
Startdeposition()
$VEL.CP = VEL_PRINT
LIN {X -1.0493,Y -9.6841,Z 59,A -2.3332,B 0.0002,C -0.0021,E1 0.1601,E2 -630.6847} C_DIS
LIN {X -2.0124,Y -9.5308,Z 59,A -2.3785,B 0.0005,C -0.0021,E1 0.1603,E2 -630.6675} C_DIS
LIN {X -3.711,Y -9.0062,Z 59,A -2.4578,B 0.0008,C -0.002,E1 0.1607,E2 -630.6269} C_DIS
LIN {X -4.5365,Y -8.6166,Z 59,A -2.5019,B 0.0009,C -0.002,E1 0.1608,E2 -630.5958} C_DIS
LIN {X -5.3249,Y -8.1567,Z 59,A -2.5573,B 0.0012,C -0.0018,E1 0.161,E2 -630.5491} C_DIS
LIN {X -6.635,Y -7.132,Z 59,A -2.6407,B 0.0014,C -0.0016,E1 0.1613,E2 -630.4692} C_DIS
LIN {X -7.251,Y -6.5046,Z 59,A -2.6867,B 0.0016,C -0.0015,E1 0.1614,E2 -630.4187} C_DIS
LIN {X -7.881,Y -5.7253,Z 59,A -2.746,B 0.0017,C -0.0013,E1 0.1616,E2 -630.3491} C_DIS
LIN {X -8.744,Y -4.2927,Z 59,A -2.8175,B 0.0019,C -0.001,E1 0.1617,E2 -630.2482} C_DIS
LIN {X -9.2435,Y -3.0727,Z 59,A -2.8918,B 0.002,C -0.0007,E1 0.1618,E2 -630.1406} C_DIS
LIN {X -9.5338,Y -1.9971,Z 59,A -2.9447,B 0.002,C -0.0005,E1 0.1619,E2 -630.053} C_DIS
LIN {X -9.7384,Y -0.2267,Z 59,A -3.0011,B 0.0021,C -0.0001,E1 0.1619,E2 -629.9297} C_DIS
LIN {X -9.6811,Y 1.0762,Z 59,A -3.0572,B 0.0021,C 0.0002,E1 0.1619,E2 -629.8171} C_DIS
LIN {X -9.4294,Y 2.4441,Z 59,A -3.0892,B 0.0021,C 0.0005,E1 0.1619,E2 -629.7187} C_DIS
LIN {X -9.0869,Y 3.5094,Z 59,A -3.1105,B 0.0021,C 0.0007,E1 0.1618,E2 -629.6404} C_DIS
LIN {X -8.6339,Y 4.5023,Z 59,A -3.1268,B 0.0019,C 0.0009,E1 0.1617,E2 -629.5659} C_DIS
LIN {X -7.8618,Y 5.7513,Z 59,A -3.1535,B 0.0017,C 0.0012,E1 0.1615,E2 -629.4589} C_DIS
LIN {X -6.7924,Y 6.9818,Z 59,A -3.1628,B 0.0015,C 0.0015,E1 0.1612,E2 -629.3588} C_DIS
LIN {X -5.5721,Y 7.9899,Z 59,A -3.1397,B 0.0013,C 0.0017,E1 0.161,E2 -629.2944} C_DIS
LIN {X -4.5602,Y 8.6075,Z 59,A -3.1284,B 0.001,C 0.0019,E1 0.1607,E2 -629.2423} C_DIS
LIN {X -3.2804,Y 9.1716,Z 59,A -3.0944,B 0.0008,C 0.0019,E1 0.1605,E2 -629.2048} C_DIS
LIN {X -2.3168,Y 9.4608,Z 59,A -3.0704,B 0.0006,C 0.0021,E1 0.1602,E2 -629.1806} C_DIS
LIN {X -1.0369,Y 9.6857,Z 59,A -3.0277,B 0.0003,C 0.0021,E1 0.16,E2 -629.1659} C_DIS
LIN {X -0.1027,Y 9.7406,Z 59,A -2.9945,B 0.0001,C 0.0021,E1 0.1598,E2 -629.1617} C_DIS
LIN {X 1.0306,Y 9.6861,Z 59,A -2.9489,B -0.0002,C 0.0021,E1 0.1595,E2 -629.1669} C_DIS
LIN {X 2.0705,Y 9.5183,Z 59,A -2.9027,B -0.0004,C 0.0021,E1 0.1593,E2 -629.181} C_DIS
LIN {X 3.1865,Y 9.2049,Z 59,A -2.8461,B -0.0007,C 0.0021,E1 0.159,E2 -629.2088} C_DIS
LIN {X 4.3518,Y 8.7147,Z 59,A -2.7833,B -0.0009,C 0.0019,E1 0.1588,E2 -629.2484} C_DIS
LIN {X 5.4635,Y 8.0644,Z 59,A -2.7164,B -0.0012,C 0.0018,E1 0.1585,E2 -629.301} C_DIS
LIN {X 6.4218,Y 7.3243,Z 59,A -2.6541,B -0.0014,C 0.0016,E1 0.1583,E2 -629.3588} C_DIS
LIN {X 7.2754,Y 6.4774,Z 59,A -2.5868,B -0.0016,C 0.0014,E1 0.1582,E2 -629.4301} C_DIS
LIN {X 7.8981,Y 5.7016,Z 59,A -2.534,B -0.0017,C 0.0013,E1 0.158,E2 -629.4928} C_DIS
LIN {X 8.4212,Y 4.8962,Z 59,A -2.4833,B -0.0018,C 0.0011,E1 0.158,E2 -629.5584} C_DIS
LIN {X 8.9452,Y 3.8561,Z 59,A -2.4287,B -0.0019,C 0.0009,E1 0.1578,E2 -629.6381} C_DIS
LIN {X 9.3531,Y 2.7212,Z 59,A -2.3692,B -0.002,C 0.0006,E1 0.1578,E2 -629.7313} C_DIS
LIN {X 9.5952,Y 1.6791,Z 59,A -2.3088,B -0.0021,C 0.0004,E1 0.1577,E2 -629.8279} C_DIS
LIN {X 9.7387,Y -0.2036,Z 59,A -2.2603,B -0.0021,C 0,E1 0.1577,E2 -629.9526} C_DIS
LIN {X 9.6701,Y -1.1722,Z 59,A -2.2113,B -0.0021,C -0.0002,E1 0.1577,E2 -630.0464} C_DIS
LIN {X 9.5022,Y -2.1421,Z 59,A -2.1884,B -0.0021,C -0.0004,E1 0.1577,E2 -630.1178} C_DIS
LIN {X 9.1815,Y -3.2533,Z 59,A -2.1741,B -0.0021,C -0.0007,E1 0.1577,E2 -630.1923} C_DIS
LIN {X 8.8501,Y -4.0689,Z 59,A -2.1421,B -0.0019,C -0.0009,E1 0.1579,E2 -630.2723} C_DIS
LIN {X 8.3436,Y -5.0269,Z 59,A -2.1304,B -0.0019,C -0.0011,E1 0.1579,E2 -630.3445} C_DIS
LIN {X 7.746,Y -5.9065,Z 59,A -2.1236,B -0.0017,C -0.0013,E1 0.1581,E2 -630.4118} C_DIS
LIN {X 7.1384,Y -6.6277,Z 59,A -2.1212,B -0.0016,C -0.0014,E1 0.1583,E2 -630.4679} C_DIS
LIN {X 6.4045,Y -7.3395,Z 59,A -2.1256,B -0.0014,C -0.0016,E1 0.1584,E2 -630.5215} C_DIS
LIN {X 5.3122,Y -8.1652,Z 59,A -2.1381,B -0.0012,C -0.0018,E1 0.1587,E2 -630.5849} C_DIS
LIN {X 4.3061,Y -8.7373,Z 59,A -2.151,B -0.0009,C -0.0019,E1 0.1589,E2 -630.6336} C_DIS
LIN {X 2.5585,Y -9.3989,Z 59,A -2.203,B -0.0006,C -0.0021,E1 0.1593,E2 -630.6739} C_DIS
LIN {X 0.9656,Y -9.693,Z 59,A -2.2541,B -0.0002,C -0.0021,E1 0.1597,E2 -630.6932} C_DIS
LIN {X -0.0615,Y -9.7408,Z 59,A -2.2923,B -0.0002,C -0.0021,E1 0.1597,E2 -630.6942} C_DIS
Enddeposition()
LIN {X -0.0615,Y -9.7408,Z 59,A -2.2923,B -0.0002,C -0.0021,E1 0.1597,E2 -630.6942} C_DIS
Startdeposition()
$VEL.CP = VEL_PRINT
LIN {X 0.4868,Y -8.7466,Z 59,A -2.2222,B -0.0002,C -0.0021,E1 0.1597,E2 -630.7013} C_DIS
LIN {X 1.6067,Y -8.6073,Z 59,A -2.189,B -0.0005,C -0.0021,E1 0.1594,E2 -630.6879} C_DIS
LIN {X 2.7508,Y -8.3169,Z 59,A -2.1624,B -0.0008,C -0.0021,E1 0.1591,E2 -630.6603} C_DIS
LIN {X 3.5728,Y -7.9983,Z 59,A -2.1502,B -0.001,C -0.0019,E1 0.1589,E2 -630.6287} C_DIS
LIN {X 4.549,Y -7.4866,Z 59,A -2.1375,B -0.0012,C -0.0018,E1 0.1586,E2 -630.5835} C_DIS
LIN {X 5.3412,Y -6.9434,Z 59,A -2.1345,B -0.0014,C -0.0016,E1 0.1584,E2 -630.5339} C_DIS
LIN {X 6.4031,Y -5.9783,Z 59,A -2.1437,B -0.0017,C -0.0014,E1 0.1582,E2 -630.4436} C_DIS
LIN {X 7.0494,Y -5.2006,Z 59,A -2.1562,B -0.0018,C -0.0012,E1 0.158,E2 -630.3733} C_DIS
LIN {X 7.633,Y -4.2988,Z 59,A -2.1724,B -0.0019,C -0.0009,E1 0.1579,E2 -630.2963} C_DIS
LIN {X 8.0263,Y -3.5027,Z 59,A -2.1936,B -0.002,C -0.0007,E1 0.1578,E2 -630.2258} C_DIS
LIN {X 8.3424,Y -2.6729,Z 59,A -2.2283,B -0.0021,C -0.0005,E1 0.1578,E2 -630.1432} C_DIS
LIN {X 8.6111,Y -1.5866,Z 59,A -2.2615,B -0.0021,C -0.0003,E1 0.1577,E2 -630.0526} C_DIS
LIN {X 8.7383,Y -0.6201,Z 59,A -2.3136,B -0.0021,C 0,E1 0.1577,E2 -629.9536} C_DIS
LIN {X 8.722,Y 0.8176,Z 59,A -2.3871,B -0.0021,C 0.0004,E1 0.1577,E2 -629.8183} C_DIS
LIN {X 8.459,Y 2.2773,Z 59,A -2.4542,B -0.0021,C 0.0007,E1 0.1577,E2 -629.6979} C_DIS
LIN {X 8.0124,Y 3.5413,Z 59,A -2.5293,B -0.0019,C 0.001,E1 0.1579,E2 -629.585} C_DIS
LIN {X 7.4134,Y 4.6611,Z 59,A -2.5777,B -0.0018,C 0.0012,E1 0.1579,E2 -629.511} C_DIS
LIN {X 6.9377,Y 5.3488,Z 59,A -2.6422,B -0.0016,C 0.0014,E1 0.1581,E2 -629.4349} C_DIS
LIN {X 6.3129,Y 6.0736,Z 59,A -2.7015,B -0.0014,C 0.0016,E1 0.1583,E2 -629.368} C_DIS
LIN {X 5.4953,Y 6.8223,Z 59,A -2.7657,B -0.0012,C 0.0018,E1 0.1585,E2 -629.3028} C_DIS
LIN {X 4.5469,Y 7.4878,Z 59,A -2.8255,B -0.001,C 0.0019,E1 0.1587,E2 -629.2504} C_DIS
LIN {X 3.3938,Y 8.0759,Z 59,A -2.8987,B -0.0006,C 0.0021,E1 0.1591,E2 -629.1958} C_DIS
LIN {X 1.7448,Y 8.5844,Z 59,A -2.9728,B -0.0003,C 0.0021,E1 0.1594,E2 -629.1623} C_DIS
LIN {X 0.7129,Y 8.7309,Z 59,A -3.0144,B 0,C 0.0021,E1 0.1597,E2 -629.1533} C_DIS
LIN {X -0.5709,Y 8.7416,Z 59,A -3.0583,B 0.0003,C 0.0021,E1 0.16,E2 -629.1572} C_DIS
LIN {X -1.4721,Y 8.6321,Z 59,A -3.0849,B 0.0005,C 0.0021,E1 0.1602,E2 -629.169} C_DIS
LIN {X -2.5809,Y 8.3713,Z 59,A -3.1079,B 0.0008,C 0.0021,E1 0.1605,E2 -629.1985} C_DIS
LIN {X -3.6101,Y 7.9813,Z 59,A -3.126,B 0.001,C 0.0019,E1 0.1607,E2 -629.2351} C_DIS
LIN {X -4.8698,Y 7.2821,Z 59,A -3.1221,B 0.0014,C 0.0017,E1 0.1611,E2 -629.315} C_DIS
LIN {X -6.3308,Y 6.054,Z 59,A -3.1261,B 0.0017,C 0.0014,E1 0.1614,E2 -629.4164} C_DIS
LIN {X -6.9775,Y 5.2959,Z 59,A -3.1073,B 0.0018,C 0.0011,E1 0.1616,E2 -629.4907} C_DIS
LIN {X -7.7296,Y 4.1209,Z 59,A -3.0846,B 0.002,C 0.0009,E1 0.1617,E2 -629.5901} C_DIS
LIN {X -8.3427,Y 2.6723,Z 59,A -3.0178,B 0.0021,C 0.0004,E1 0.1619,E2 -629.7397} C_DIS
LIN {X -8.6886,Y 1.1176,Z 59,A -2.9713,B 0.0021,C 0.0001,E1 0.1619,E2 -629.8639} C_DIS
LIN {X -8.7597,Y -0.1063,Z 59,A -2.9186,B 0.0021,C -0.0002,E1 0.1619,E2 -629.9704} C_DIS
LIN {X -8.6177,Y -1.5735,Z 59,A -2.8608,B 0.0021,C -0.0005,E1 0.1619,E2 -630.0847} C_DIS
LIN {X -8.4064,Y -2.4534,Z 59,A -2.8167,B 0.0021,C -0.0007,E1 0.1619,E2 -630.1582} C_DIS
LIN {X -8.0566,Y -3.4398,Z 59,A -2.7542,B 0.0019,C -0.001,E1 0.1618,E2 -630.2496} C_DIS
Enddeposition()
END
